C01824=1205.778,287.923,-66.895,-176.683,7.105,148.360
C01825=1205.774,288.171,-66.924,-176.680,7.108,148.360
C01826=1205.769,288.419,-66.953,-176.678,7.110,148.360
C01827=1205.765,288.694,-66.985,-176.675,7.113,148.360
C01828=1205.760,288.968,-67.017,-176.672,7.116,148.360
C01829=1205.756,289.243,-67.049,-176.670,7.119,148.360
C01830=1205.750,289.517,-67.081,-176.667,7.122,148.360
C01831=1205.747,289.765,-67.110,-176.664,7.124,148.359
C01832=1205.742,290.013,-67.139,-176.662,7.127,148.359
C01833=1205.738,290.261,-67.168,-176.660,7.129,148.359
C01834=1205.733,290.510,-67.197,-176.657,7.132,148.359
C01835=1205.729,290.758,-67.226,-176.655,7.134,148.359
C01836=1205.725,291.006,-67.256,-176.652,7.137,148.359
C01837=1205.720,291.255,-67.284,-176.650,7.139,148.359
C01838=1205.715,291.503,-67.314,-176.647,7.142,148.359
C01839=1205.712,291.751,-67.342,-176.645,7.144,148.359
C01840=1205.708,291.999,-67.372,-176.642,7.147,148.359
C01841=1205.703,292.248,-67.401,-176.640,7.149,148.359
C01842=1205.699,292.496,-67.430,-176.637,7.152,148.359
C01843=1205.694,292.744,-67.459,-176.635,7.154,148.359
C01844=1205.690,292.992,-67.489,-176.632,7.158,148.359
C01845=1205.686,293.240,-67.518,-176.630,7.160,148.359
C01846=1205.682,293.489,-67.547,-176.627,7.162,148.358
C01847=1205.677,293.737,-67.576,-176.624,7.165,148.358
C01848=1205.673,293.985,-67.605,-176.622,7.168,148.358
C01849=1205.668,294.233,-67.635,-176.620,7.171,148.358
C01850=1205.664,294.482,-67.664,-176.617,7.173,148.358
C01851=1205.660,294.730,-67.694,-176.615,7.176,148.358
C01852=1205.656,294.978,-67.723,-176.613,7.178,148.358
C01853=1205.651,295.227,-67.752,-176.610,7.181,148.358
C01854=1205.647,295.475,-67.781,-176.608,7.183,148.358
C01855=1205.642,295.723,-67.810,-176.605,7.186,148.358
C01856=1205.638,295.971,-67.840,-176.603,7.189,148.358
C01857=1205.634,296.219,-67.869,-176.600,7.191,148.358
C01858=1205.630,296.468,-67.899,-176.597,7.194,148.358
C01859=1205.626,296.716,-67.928,-176.595,7.196,148.358
C01860=1205.621,296.964,-67.958,-176.592,7.199,148.358
C01861=1205.617,297.213,-67.987,-176.590,7.202,148.357
C01862=1205.613,297.461,-68.017,-176.588,7.205,148.357
C01863=1205.608,297.709,-68.047,-176.585,7.207,148.357
C01864=1205.603,297.957,-68.076,-176.583,7.210,148.357
C01865=1205.599,298.205,-68.105,-176.581,7.212,148.357
C01866=1205.595,298.453,-68.135,-176.578,7.215,148.357
C01867=1205.591,298.702,-68.164,-176.575,7.218,148.357
C01868=1205.587,298.950,-68.194,-176.573,7.220,148.357
C01869=1205.583,299.198,-68.224,-176.570,7.223,148.357
C01870=1205.579,299.446,-68.253,-176.568,7.226,148.357
C01871=1205.574,299.694,-68.283,-176.566,7.229,148.357
C01872=1205.570,299.943,-68.313,-176.563,7.231,148.357
C01873=1205.565,300.191,-68.342,-176.561,7.234,148.357
C01874=1205.561,300.439,-68.372,-176.558,7.237,148.357
C01875=1205.557,300.688,-68.401,-176.556,7.239,148.357
C01876=1205.553,300.935,-68.431,-176.553,7.242,148.357
C01877=1205.548,301.184,-68.461,-176.551,7.244,148.357
C01878=1205.544,301.432,-68.491,-176.548,7.247,148.357
C01879=1205.540,301.680,-68.520,-176.546,7.249,148.357
C01880=1205.536,301.929,-68.550,-176.544,7.252,148.357
C01881=1205.531,302.177,-68.580,-176.541,7.256,148.357
C01882=1205.527,302.425,-68.610,-176.539,7.258,148.357
C01883=1205.523,302.673,-68.639,-176.536,7.261,148.357
C01884=1205.518,302.921,-68.669,-176.534,7.263,148.357
C01885=1205.514,303.169,-68.700,-176.531,7.266,148.357
C01886=1205.510,303.418,-68.729,-176.529,7.268,148.357
C01887=1205.506,303.666,-68.758,-176.526,7.271,148.357
C01888=1205.501,303.914,-68.789,-176.524,7.274,148.357
C01889=1205.497,304.162,-68.819,-176.522,7.276,148.357
C01890=1205.493,304.410,-68.848,-176.519,7.279,148.356
C01891=1205.488,304.658,-68.879,-176.517,7.282,148.356
C01892=1205.484,304.907,-68.908,-176.514,7.285,148.356
C01893=1205.480,305.154,-68.939,-176.511,7.288,148.356
C01894=1205.475,305.403,-68.969,-176.509,7.290,148.356
C01895=1205.471,305.651,-68.998,-176.507,7.293,148.356
C01896=1205.467,305.899,-69.028,-176.505,7.295,148.356
C01897=1205.462,306.147,-69.058,-176.502,7.298,148.356
C01898=1205.458,306.395,-69.088,-176.500,7.301,148.356
C01899=1205.454,306.643,-69.118,-176.497,7.304,148.356
C01900=1205.449,306.891,-69.149,-176.495,7.307,148.356
C01901=1205.445,307.139,-69.178,-176.493,7.309,148.356
C01902=1205.441,307.388,-69.209,-176.490,7.312,148.356
C01903=1205.437,307.636,-69.239,-176.488,7.314,148.356
C01904=1205.433,307.884,-69.269,-176.485,7.317,148.356
C01905=1205.428,308.133,-69.299,-176.482,7.320,148.356
C01906=1205.424,308.380,-69.329,-176.480,7.322,148.356
C01907=1205.419,308.629,-69.359,-176.478,7.325,148.356
C01908=1205.415,308.876,-69.389,-176.475,7.329,148.356
C01909=1205.411,309.125,-69.419,-176.473,7.331,148.356
C01910=1205.407,309.373,-69.449,-176.471,7.334,148.356
C01911=1205.403,309.621,-69.481,-176.469,7.336,148.356
C01912=1205.398,309.870,-69.510,-176.466,7.339,148.356
C01913=1205.394,310.118,-69.541,-176.463,7.342,148.356
C01914=1205.390,310.365,-69.571,-176.461,7.344,148.356
C01915=1205.385,310.614,-69.601,-176.458,7.347,148.356
C01916=1205.381,310.861,-69.631,-176.457,7.350,148.356
C01917=1205.377,311.110,-69.662,-176.454,7.353,148.356
C01918=1205.373,311.358,-69.692,-176.451,7.356,148.356
C01919=1205.368,311.606,-69.723,-176.449,7.358,148.356
C01920=1205.365,311.854,-69.753,-176.446,7.361,148.356
C01921=1205.360,312.103,-69.783,-176.444,7.363,148.356
C01922=1205.356,312.350,-69.813,-176.442,7.367,148.356
C01923=1205.352,312.599,-69.844,-176.439,7.370,148.356
C01924=1205.347,312.847,-69.875,-176.437,7.372,148.356
C01925=1205.343,313.094,-69.905,-176.435,7.375,148.356
C01926=1205.338,313.343,-69.935,-176.432,7.378,148.356
C01927=1205.334,313.591,-69.965,-176.430,7.381,148.357
C01928=1205.330,313.839,-69.996,-176.428,7.384,148.357
C01929=1205.326,314.087,-70.027,-176.425,7.386,148.356
C01930=1205.322,314.335,-70.057,-176.423,7.389,148.356
C01931=1205.317,314.611,-70.091,-176.420,7.392,148.356
C01932=1205.312,314.887,-70.125,-176.418,7.395,148.357
C01933=1205.308,315.164,-70.159,-176.415,7.398,148.357
C01934=1205.303,315.440,-70.193,-176.413,7.401,148.357
C01935=1205.298,315.688,-70.224,-176.410,7.404,148.357
C01936=1205.294,315.936,-70.254,-176.408,7.406,148.357
C01937=1205.290,316.184,-70.285,-176.406,7.410,148.357
C01938=1205.286,316.432,-70.316,-176.403,7.413,148.357
C01939=1205.282,316.680,-70.346,-176.401,7.415,148.357
C01940=1205.277,316.928,-70.377,-176.398,7.418,148.357
C01941=1205.273,317.177,-70.408,-176.396,7.421,148.357
C01942=1205.269,317.424,-70.438,-176.394,7.424,148.357
C01943=1205.265,317.672,-70.469,-176.391,7.427,148.357
C01944=1205.261,317.921,-70.500,-176.389,7.429,148.357
C01945=1205.256,318.169,-70.531,-176.387,7.432,148.357
C01946=1205.252,318.416,-70.561,-176.384,7.435,148.357
C01947=1205.248,318.665,-70.592,-176.382,7.437,148.357
C01948=1205.244,318.913,-70.623,-176.380,7.441,148.357
C01949=1205.239,319.161,-70.654,-176.377,7.444,148.357
C01950=1205.236,319.409,-70.684,-176.375,7.446,148.357
C01951=1205.231,319.657,-70.715,-176.373,7.449,148.357
C01952=1205.226,319.905,-70.746,-176.370,7.452,148.357
C01953=1205.222,320.154,-70.777,-176.368,7.455,148.357
C01954=1205.218,320.401,-70.809,-176.365,7.458,148.357
C01955=1205.214,320.649,-70.839,-176.363,7.460,148.357
C01956=1205.210,320.898,-70.870,-176.361,7.463,148.357
C01957=1205.206,321.145,-70.901,-176.359,7.466,148.358
C01958=1205.201,321.393,-70.931,-176.356,7.469,148.358
C01959=1205.197,321.641,-70.963,-176.354,7.472,148.358
C01960=1205.193,321.889,-70.994,-176.352,7.475,148.358
C01961=1205.188,322.137,-71.025,-176.349,7.477,148.358
C01962=1205.185,322.386,-71.055,-176.347,7.480,148.358
C01963=1205.180,322.633,-71.087,-176.345,7.483,148.358
C01964=1205.176,322.882,-71.118,-176.342,7.486,148.358
C01965=1205.172,323.130,-71.149,-176.340,7.489,148.358
C01966=1205.167,323.378,-71.179,-176.338,7.491,148.358
C01967=1205.164,323.626,-71.211,-176.335,7.494,148.358
C01968=1205.159,323.874,-71.242,-176.333,7.498,148.358
C01969=1205.155,324.122,-71.273,-176.331,7.500,148.358
C01970=1205.151,324.370,-71.305,-176.329,7.503,148.359
C01971=1205.147,324.618,-71.336,-176.326,7.506,148.359
C01972=1205.142,324.866,-71.367,-176.324,7.509,148.358
C01973=1205.138,325.114,-71.398,-176.322,7.512,148.359
C01974=1205.134,325.362,-71.429,-176.319,7.515,148.359
C01975=1205.130,325.609,-71.460,-176.317,7.517,148.359
C01976=1205.126,325.858,-71.491,-176.315,7.520,148.359
C01977=1205.121,326.106,-71.522,-176.313,7.523,148.359
C01978=1205.118,326.354,-71.554,-176.310,7.526,148.359
C01979=1205.113,326.602,-71.585,-176.308,7.529,148.359
C01980=1205.109,326.850,-71.616,-176.306,7.531,148.359
C01981=1205.105,327.098,-71.647,-176.303,7.535,148.359
C01982=1205.100,327.346,-71.679,-176.301,7.538,148.359
C01983=1205.096,327.594,-71.710,-176.299,7.540,148.359
C01984=1205.091,327.842,-71.742,-176.297,7.543,148.360
C01985=1205.087,328.090,-71.773,-176.294,7.546,148.360
C01986=1205.083,328.338,-71.804,-176.293,7.549,148.360
C01987=1205.079,328.586,-71.836,-176.290,7.552,148.360
C01988=1205.075,328.834,-71.867,-176.288,7.555,148.360
C01989=1205.071,329.082,-71.898,-176.285,7.558,148.360
C01990=1205.067,329.330,-71.930,-176.283,7.561,148.360
C01991=1205.063,329.578,-71.961,-176.282,7.563,148.360
C01992=1205.058,329.826,-71.992,-176.279,7.566,148.360
C01993=1205.054,330.074,-72.024,-176.277,7.570,148.361
C01994=1205.050,330.323,-72.056,-176.275,7.572,148.360
C01995=1205.045,330.570,-72.087,-176.272,7.575,148.361
C01996=1205.042,330.818,-72.119,-176.270,7.578,148.361
C01997=1205.037,331.066,-72.150,-176.268,7.581,148.361
C01998=1205.033,331.314,-72.182,-176.265,7.584,148.361
C01999=1205.029,331.561,-72.213,-176.263,7.587,148.361
C02000=1205.025,331.810,-72.244,-176.261,7.590,148.361
C02001=1205.020,332.058,-72.276,-176.259,7.593,148.361
C02002=1205.016,332.306,-72.308,-176.257,7.596,148.362
C02003=1205.012,332.553,-72.340,-176.254,7.598,148.361
C02004=1205.008,332.802,-72.371,-176.252,7.602,148.362
C02005=1205.004,333.050,-72.403,-176.251,7.604,148.362
C02006=1204.999,333.297,-72.435,-176.248,7.607,148.362
C02007=1204.996,333.545,-72.467,-176.246,7.611,148.362
C02008=1204.991,333.793,-72.498,-176.244,7.613,148.362
C02009=1204.987,334.041,-72.529,-176.241,7.616,148.362
C02010=1204.983,334.290,-72.562,-176.239,7.619,148.362
C02011=1204.978,334.537,-72.593,-176.237,7.622,148.362
C02012=1204.975,334.785,-72.625,-176.235,7.625,148.363
C02013=1204.970,335.032,-72.657,-176.233,7.628,148.363
C02014=1204.966,335.281,-72.689,-176.230,7.631,148.363
C02015=1204.962,335.529,-72.720,-176.228,7.634,148.363
C02016=1204.958,335.777,-72.752,-176.226,7.637,148.363
C02017=1204.953,336.025,-72.784,-176.224,7.640,148.363
C02018=1204.950,336.273,-72.816,-176.222,7.643,148.363
C02019=1204.945,336.520,-72.847,-176.220,7.645,148.364
C02020=1204.941,336.769,-72.880,-176.218,7.649,148.364
C02021=1204.936,337.016,-72.911,-176.215,7.652,148.364
C02022=1204.933,337.264,-72.943,-176.213,7.654,148.364
C02023=1204.928,337.513,-72.976,-176.211,7.657,148.364
C02024=1204.924,337.760,-73.007,-176.209,7.661,148.364
C02025=1204.920,338.008,-73.039,-176.207,7.663,148.364
C02026=1204.916,338.256,-73.071,-176.205,7.666,148.365
C02027=1204.912,338.504,-73.103,-176.202,7.670,148.365
C02028=1204.908,338.752,-73.135,-176.201,7.672,148.365
C02029=1204.903,339.000,-73.167,-176.198,7.675,148.365
C02030=1204.900,339.248,-73.199,-176.196,7.678,148.365
C02031=1204.895,339.496,-73.231,-176.194,7.681,148.365
C02032=1204.891,339.744,-73.263,-176.192,7.684,148.366
C02033=1204.887,339.992,-73.295,-176.190,7.687,148.366
C02034=1204.883,340.239,-73.327,-176.188,7.690,148.366
C02035=1204.878,340.518,-73.363,-176.186,7.693,148.366
C02036=1204.873,340.795,-73.399,-176.183,7.697,148.366
C02037=1204.869,341.074,-73.435,-176.181,7.700,148.367
C02038=1204.864,341.353,-73.471,-176.179,7.703,148.367
C02039=1204.860,341.600,-73.504,-176.177,7.707,148.367
C02040=1204.856,341.848,-73.536,-176.174,7.710,148.367
C02041=1204.851,342.096,-73.567,-176.172,7.712,148.367
C02042=1204.847,342.344,-73.600,-176.170,7.716,148.367
C02043=1204.843,342.592,-73.632,-176.168,7.718,148.368
C02044=1204.839,342.840,-73.665,-176.166,7.721,148.368
C02045=1204.835,343.087,-73.696,-176.164,7.725,148.368
C02046=1204.830,343.335,-73.729,-176.162,7.727,148.368
C02047=1204.826,343.584,-73.761,-176.160,7.731,148.368
C02048=1204.823,343.831,-73.794,-176.158,7.734,148.369
C02049=1204.818,344.079,-73.826,-176.156,7.736,148.369
C02050=1204.814,344.327,-73.858,-176.154,7.739,148.369
C02051=1204.810,344.575,-73.891,-176.151,7.743,148.369
C02052=1204.806,344.823,-73.923,-176.150,7.745,148.369
C02053=1204.802,345.071,-73.955,-176.147,7.749,148.369
C02054=1204.797,345.318,-73.988,-176.146,7.751,148.370
C02055=1204.793,345.566,-74.020,-176.144,7.755,148.370
C02056=1204.789,345.814,-74.052,-176.141,7.758,148.370
C02057=1204.785,346.062,-74.085,-176.140,7.760,148.370
C02058=1204.781,346.310,-74.117,-176.137,7.764,148.370
C02059=1204.776,346.557,-74.150,-176.136,7.766,148.371
C02060=1204.772,346.805,-74.182,-176.134,7.770,148.371
C02061=1204.768,347.054,-74.214,-176.131,7.773,148.371
C02062=1204.764,347.301,-74.247,-176.130,7.775,148.371
C02063=1204.760,347.549,-74.279,-176.128,7.779,148.371
C02064=1204.755,347.796,-74.312,-176.125,7.782,148.372
C02065=1204.751,348.045,-74.345,-176.124,7.785,148.372
C02066=1204.747,348.292,-74.377,-176.121,7.788,148.372
C02067=1204.743,348.541,-74.410,-176.120,7.790,148.372
C02068=1204.739,348.788,-74.443,-176.118,7.794,148.373
C02069=1204.735,349.036,-74.475,-176.116,7.797,148.373
C02070=1204.731,349.284,-74.508,-176.114,7.800,148.373
C02071=1204.726,349.532,-74.540,-176.112,7.803,148.373
C02072=1204.723,349.779,-74.572,-176.110,7.806,148.374
C02073=1204.718,350.027,-74.605,-176.108,7.809,148.374
C02074=1204.714,350.275,-74.638,-176.106,7.813,148.374
C02075=1204.710,350.523,-74.671,-176.104,7.815,148.374
C02076=1204.706,350.771,-74.703,-176.102,7.818,148.374
C02077=1204.702,351.019,-74.736,-176.101,7.821,148.375
C02078=1204.698,351.267,-74.769,-176.099,7.825,148.375
C02079=1204.693,351.515,-74.802,-176.096,7.828,148.375
C02080=1204.690,351.762,-74.834,-176.095,7.830,148.375
C02081=1204.685,352.010,-74.866,-176.092,7.834,148.376
C02082=1204.681,352.258,-74.900,-176.091,7.836,148.376
C02083=1204.677,352.505,-74.933,-176.089,7.840,148.376
C02084=1204.672,352.754,-74.965,-176.087,7.843,148.376
C02085=1204.669,353.001,-74.998,-176.085,7.846,148.377
C02086=1204.665,353.249,-75.031,-176.083,7.849,148.377
C02087=1204.661,353.496,-75.064,-176.082,7.852,148.377
C02088=1204.656,353.745,-75.096,-176.079,7.855,148.377
C02089=1204.652,353.993,-75.130,-176.077,7.859,148.378
C02090=1204.648,354.240,-75.163,-176.076,7.861,148.378
C02091=1204.645,354.488,-75.195,-176.074,7.865,148.378
C02092=1204.640,354.736,-75.228,-176.072,7.867,148.379
C02093=1204.636,354.984,-75.261,-176.070,7.871,148.379
C02094=1204.632,355.232,-75.294,-176.068,7.874,148.379
C02095=1204.628,355.479,-75.327,-176.067,7.877,148.379
C02096=1204.624,355.727,-75.360,-176.064,7.880,148.380
C02097=1204.619,355.975,-75.394,-176.063,7.883,148.380
C02098=1204.615,356.223,-75.426,-176.061,7.886,148.380
C02099=1204.611,356.471,-75.459,-176.059,7.889,148.380
C02100=1204.607,356.718,-75.492,-176.057,7.892,148.381
C02101=1204.603,356.966,-75.525,-176.055,7.896,148.381
C02102=1204.599,357.214,-75.558,-176.054,7.898,148.381
C02103=1204.595,357.461,-75.591,-176.052,7.902,148.382
C02104=1204.591,357.709,-75.624,-176.050,7.904,148.382
C02105=1204.587,357.957,-75.657,-176.048,7.908,148.382
C02106=1204.583,358.205,-75.691,-176.047,7.910,148.382
C02107=1204.578,358.452,-75.724,-176.045,7.914,148.383
C02108=1204.574,358.700,-75.757,-176.043,7.917,148.383
C02109=1204.570,358.948,-75.790,-176.041,7.920,148.383
C02110=1204.566,359.195,-75.823,-176.039,7.924,148.384
C02111=1204.562,359.443,-75.856,-176.038,7.926,148.384
C02112=1204.558,359.691,-75.890,-176.036,7.930,148.384
C02113=1204.554,359.939,-75.923,-176.034,7.932,148.385
C02114=1204.549,360.186,-75.956,-176.032,7.936,148.385
C02115=1204.545,360.434,-75.989,-176.031,7.938,148.385
C02116=1204.541,360.682,-76.022,-176.029,7.942,148.386
C02117=1204.537,360.930,-76.055,-176.027,7.945,148.386
C02118=1204.533,361.177,-76.088,-176.026,7.948,148.386
C02119=1204.529,361.425,-76.122,-176.024,7.951,148.386
C02120=1204.525,361.673,-76.155,-176.022,7.954,148.387
C02121=1204.521,361.921,-76.188,-176.021,7.957,148.387
C02122=1204.517,362.169,-76.221,-176.019,7.961,148.387
C02123=1204.513,362.417,-76.255,-176.018,7.963,148.388
C02124=1204.509,362.664,-76.288,-176.015,7.967,148.388
C02125=1204.505,362.912,-76.322,-176.014,7.970,148.388
C02126=1204.500,363.160,-76.355,-176.012,7.973,148.389
C02127=1204.496,363.407,-76.389,-176.011,7.976,148.389
C02128=1204.492,363.655,-76.422,-176.009,7.979,148.390
C02129=1204.488,363.903,-76.455,-176.007,7.982,148.390
C02130=1204.484,364.151,-76.489,-176.006,7.985,148.390
C02131=1204.480,364.398,-76.522,-176.004,7.988,148.391
C02132=1204.476,364.646,-76.555,-176.002,7.992,148.391
C02133=1204.472,364.894,-76.589,-176.001,7.994,148.391
C02134=1204.467,365.141,-76.623,-175.999,7.998,148.392
C02135=1204.463,365.389,-76.656,-175.998,8.001,148.392
C02136=1204.459,365.637,-76.689,-175.996,8.003,148.392
C02137=1204.456,365.885,-76.723,-175.995,8.007,148.393
C02138=1204.452,366.132,-76.757,-175.993,8.010,148.393
C02139=1204.447,366.413,-76.795,-175.992,8.013,148.393
C02140=1204.442,366.693,-76.832,-175.990,8.017,148.394
C02141=1204.437,366.974,-76.871,-175.988,8.021,148.394
C02142=1204.433,367.254,-76.908,-175.986,8.024,148.395
C02143=1204.428,367.502,-76.942,-175.985,8.027,148.395
C02144=1204.424,367.750,-76.975,-175.983,8.031,148.395
C02145=1204.421,367.997,-77.010,-175.982,8.033,148.396
C02146=1204.417,368.245,-77.043,-175.980,8.036,148.396
C02147=1204.412,368.493,-77.077,-175.979,8.040,148.397
C02148=1204.408,368.740,-77.110,-175.977,8.043,148.397
C02149=1204.404,368.988,-77.144,-175.976,8.045,148.397
C02150=1204.401,369.236,-77.178,-175.974,8.049,148.398
C02151=1204.396,369.484,-77.211,-175.973,8.052,148.398
C02152=1204.392,369.731,-77.245,-175.972,8.054,148.398
C02153=1204.388,369.979,-77.279,-175.970,8.058,148.399
C02154=1204.384,370.226,-77.312,-175.969,8.061,148.399
C02155=1204.380,370.475,-77.347,-175.967,8.064,148.400
C02156=1204.376,370.722,-77.380,-175.966,8.067,148.400
C02157=1204.372,370.969,-77.414,-175.964,8.070,148.400
C02158=1204.367,371.217,-77.447,-175.963,8.073,148.401
C02159=1204.364,371.465,-77.482,-175.962,8.076,148.401
C02160=1204.360,371.713,-77.515,-175.960,8.079,148.402
C02161=1204.355,371.960,-77.549,-175.959,8.082,148.402
C02162=1204.351,372.208,-77.583,-175.958,8.085,148.402
C02163=1204.347,372.455,-77.616,-175.956,8.089,148.403
C02164=1204.343,372.703,-77.651,-175.955,8.092,148.404
C02165=1204.339,372.951,-77.684,-175.954,8.095,148.404
C02166=1204.335,373.198,-77.718,-175.953,8.097,148.404
C02167=1204.331,373.447,-77.752,-175.952,8.100,148.405
C02168=1204.327,373.694,-77.786,-175.950,8.104,148.405
C02169=1204.323,373.941,-77.820,-175.949,8.107,148.406
C02170=1204.318,374.189,-77.854,-175.947,8.109,148.406
C02171=1204.315,374.437,-77.888,-175.946,8.112,148.406
C02172=1204.310,374.685,-77.922,-175.945,8.115,148.407
C02173=1204.306,374.932,-77.956,-175.944,8.119,148.407
C02174=1204.303,375.179,-77.989,-175.942,8.122,148.408
C02175=1204.298,375.428,-78.023,-175.941,8.125,148.408
C02176=1204.295,375.675,-78.057,-175.940,8.127,148.408
C02177=1204.290,375.923,-78.092,-175.939,8.130,148.409
C02178=1204.286,376.171,-78.125,-175.938,8.133,148.409
C02179=1204.283,376.418,-78.159,-175.936,8.137,148.410
C02180=1204.278,376.666,-78.194,-175.935,8.140,148.410
C02181=1204.275,376.913,-78.228,-175.934,8.143,148.411
C02182=1204.270,377.161,-78.262,-175.933,8.146,148.411
C02183=1204.266,377.408,-78.296,-175.932,8.148,148.412
C02184=1204.262,377.656,-78.330,-175.931,8.151,148.412
C02185=1204.258,377.904,-78.364,-175.930,8.154,148.413
C02186=1204.253,378.152,-78.398,-175.929,8.157,148.413
C02187=1204.250,378.399,-78.432,-175.928,8.160,148.413
C02188=1204.246,378.647,-78.467,-175.927,8.163,148.414
C02189=1204.242,378.894,-78.501,-175.926,8.166,148.414
C02190=1204.237,379.142,-78.534,-175.924,8.170,148.415
C02191=1204.234,379.390,-78.569,-175.923,8.173,148.415
C02192=1204.229,379.637,-78.603,-175.922,8.175,148.416
C02193=1204.225,379.884,-78.637,-175.921,8.178,148.416
C02194=1204.221,380.133,-78.672,-175.920,8.181,148.417
C02195=1204.217,380.380,-78.705,-175.919,8.184,148.417
C02196=1204.213,380.628,-78.739,-175.918,8.187,148.418
C02197=1204.209,380.876,-78.774,-175.917,8.190,148.418
C02198=1204.205,381.123,-78.808,-175.916,8.193,148.419
C02199=1204.202,381.371,-78.842,-175.915,8.196,148.419
C02200=1204.197,381.618,-78.877,-175.913,8.199,148.420
C02201=1204.193,381.865,-78.911,-175.913,8.201,148.420
C02202=1204.189,382.113,-78.945,-175.912,8.204,148.421
C02203=1204.184,382.361,-78.979,-175.911,8.207,148.421
C02204=1204.180,382.609,-79.013,-175.910,8.210,148.421
C02205=1204.177,382.857,-79.048,-175.909,8.213,148.422
C02206=1204.173,383.104,-79.082,-175.908,8.216,148.422
C02207=1204.169,383.352,-79.117,-175.907,8.219,148.423
C02208=1204.164,383.599,-79.151,-175.906,8.222,148.423
C02209=1204.160,383.846,-79.185,-175.905,8.225,148.424
C02210=1204.156,384.095,-79.220,-175.904,8.228,148.424
C02211=1204.153,384.342,-79.254,-175.904,8.230,148.425
C02212=1204.149,384.590,-79.289,-175.903,8.233,148.425
C02213=1204.144,384.837,-79.323,-175.902,8.236,148.426
C02214=1204.140,385.084,-79.357,-175.901,8.239,148.427
C02215=1204.136,385.332,-79.392,-175.900,8.242,148.427
C02216=1204.132,385.580,-79.426,-175.899,8.245,148.428
C02217=1204.128,385.828,-79.460,-175.898,8.247,148.428
C02218=1204.124,386.075,-79.495,-175.898,8.250,148.428
C02219=1204.120,386.322,-79.529,-175.897,8.253,148.429
C02220=1204.116,386.570,-79.564,-175.896,8.256,148.429
C02221=1204.111,386.818,-79.598,-175.895,8.259,148.430
C02222=1204.108,387.066,-79.632,-175.894,8.261,148.430
C02223=1204.104,387.313,-79.667,-175.894,8.264,148.431
C02224=1204.100,387.561,-79.702,-175.893,8.267,148.432
C02225=1204.096,387.808,-79.735,-175.892,8.269,148.432
C02226=1204.092,388.056,-79.771,-175.891,8.272,148.432
C02227=1204.088,388.303,-79.805,-175.891,8.275,148.433
C02228=1204.084,388.550,-79.839,-175.889,8.278,148.433
C02229=1204.080,388.798,-79.874,-175.889,8.280,148.434
C02230=1204.075,389.046,-79.909,-175.888,8.283,148.435
C02231=1204.072,389.294,-79.943,-175.887,8.286,148.435
C02232=1204.067,389.541,-79.977,-175.887,8.288,148.436
C02233=1204.063,389.789,-80.012,-175.886,8.292,148.436
C02234=1204.059,390.037,-80.047,-175.885,8.295,148.437
C02235=1204.056,390.284,-80.082,-175.885,8.297,148.437
C02236=1204.051,390.531,-80.116,-175.884,8.300,148.438
C02237=1204.047,390.779,-80.151,-175.884,8.302,148.438
C02238=1204.044,391.026,-80.185,-175.883,8.305,148.439
C02239=1204.040,391.275,-80.220,-175.882,8.308,148.439
C02240=1204.035,391.522,-80.254,-175.882,8.310,148.440
C02241=1204.031,391.769,-80.290,-175.881,8.313,148.440
C02242=1204.028,392.017,-80.323,-175.880,8.315,148.441
C02243=1204.022,392.300,-80.363,-175.879,8.318,148.441
C02244=1204.018,392.582,-80.403,-175.879,8.321,148.442
C02245=1204.013,392.865,-80.442,-175.878,8.325,148.442
C02246=1204.009,393.148,-80.482,-175.877,8.328,148.443
C02247=1204.005,393.395,-80.516,-175.877,8.330,148.444
C02248=1204.001,393.642,-80.552,-175.876,8.333,148.444
C02249=1203.997,393.890,-80.586,-175.876,8.335,148.445
C02250=1203.993,394.138,-80.621,-175.875,8.338,148.445
C02251=1203.988,394.385,-80.655,-175.874,8.340,148.446
C02252=1203.985,394.633,-80.691,-175.874,8.344,148.446
C02253=1203.980,394.880,-80.725,-175.873,8.346,148.447
C02254=1203.977,395.128,-80.759,-175.873,8.349,148.447
C02255=1203.972,395.375,-80.794,-175.872,8.351,148.448
C02256=1203.969,395.623,-80.829,-175.871,8.354,148.448
C02257=1203.964,395.870,-80.864,-175.871,8.356,148.449
C02258=1203.960,396.118,-80.899,-175.871,8.359,148.449
C02259=1203.957,396.365,-80.933,-175.870,8.362,148.450
C02260=1203.953,396.613,-80.968,-175.869,8.364,148.450
C02261=1203.949,396.861,-81.003,-175.869,8.367,148.451
C02262=1203.945,397.108,-81.038,-175.868,8.369,148.451
C02263=1203.941,397.356,-81.073,-175.868,8.371,148.452
C02264=1203.936,397.603,-81.107,-175.867,8.374,148.452
C02265=1203.933,397.851,-81.142,-175.867,8.376,148.453
C02266=1203.928,398.098,-81.177,-175.866,8.379,148.453
C02267=1203.925,398.346,-81.212,-175.866,8.382,148.454
C02268=1203.920,398.593,-81.247,-175.865,8.384,148.454
C02269=1203.916,398.841,-81.282,-175.865,8.387,148.455
C02270=1203.912,399.088,-81.317,-175.864,8.389,148.456
C02271=1203.908,399.336,-81.352,-175.864,8.391,148.456
C02272=1203.905,399.584,-81.386,-175.864,8.394,148.456
C02273=1203.901,399.831,-81.421,-175.863,8.397,148.457
C02274=1203.897,400.079,-81.456,-175.863,8.399,148.458
C02275=1203.892,400.325,-81.491,-175.862,8.401,148.458
C02276=1203.888,400.574,-81.526,-175.862,8.404,148.459
C02277=1203.884,400.821,-81.560,-175.861,8.406,148.459
C02278=1203.880,401.068,-81.596,-175.861,8.409,148.460
C02279=1203.876,401.316,-81.630,-175.860,8.411,148.460
C02280=1203.872,401.563,-81.666,-175.860,8.414,148.461
C02281=1203.869,401.811,-81.700,-175.859,8.416,148.461
C02282=1203.864,402.058,-81.735,-175.859,8.418,148.462
C02283=1203.860,402.306,-81.770,-175.859,8.420,148.462
C02284=1203.856,402.553,-81.805,-175.858,8.423,148.463
C02285=1203.852,402.801,-81.840,-175.858,8.426,148.463
C02286=1203.848,403.049,-81.875,-175.857,8.428,148.464
C02287=1203.844,403.296,-81.910,-175.857,8.430,148.464
C02288=1203.840,403.544,-81.945,-175.856,8.432,148.465
C02289=1203.836,403.791,-81.980,-175.856,8.435,148.465
C02290=1203.832,404.039,-82.015,-175.855,8.438,148.466
C02291=1203.827,404.286,-82.050,-175.855,8.440,148.466
C02292=1203.824,404.534,-82.085,-175.855,8.442,148.467
C02293=1203.820,404.781,-82.121,-175.855,8.444,148.467
C02294=1203.816,405.028,-82.156,-175.854,8.446,148.468
C02295=1203.812,405.276,-82.191,-175.854,8.449,148.468
C02296=1203.809,405.524,-82.226,-175.854,8.451,148.469
C02297=1203.804,405.771,-82.260,-175.853,8.454,148.469
C02298=1203.800,406.018,-82.296,-175.853,8.456,148.470
C02299=1203.796,406.266,-82.330,-175.853,8.459,148.470
C02300=1203.792,406.513,-82.366,-175.852,8.461,148.471
C02301=1203.788,406.762,-82.400,-175.852,8.463,148.471
C02302=1203.784,407.008,-82.436,-175.851,8.465,148.472
C02303=1203.780,407.256,-82.470,-175.851,8.467,148.472
C02304=1203.776,407.503,-82.506,-175.851,8.470,148.473
C02305=1203.772,407.751,-82.541,-175.850,8.472,148.473
C02306=1203.768,407.999,-82.576,-175.850,8.474,148.474
C02307=1203.764,408.246,-82.611,-175.850,8.476,148.474
C02308=1203.760,408.494,-82.646,-175.850,8.478,148.475
C02309=1203.756,408.741,-82.682,-175.849,8.481,148.475
C02310=1203.752,408.988,-82.717,-175.848,8.484,148.476
C02311=1203.748,409.236,-82.752,-175.848,8.486,148.476
C02312=1203.744,409.484,-82.787,-175.848,8.488,148.477
C02313=1203.740,409.731,-82.822,-175.847,8.490,148.477
C02314=1203.736,409.979,-82.857,-175.847,8.493,148.478
C02315=1203.732,410.225,-82.892,-175.847,8.495,148.478
C02316=1203.728,410.474,-82.927,-175.846,8.497,148.479
C02317=1203.724,410.721,-82.963,-175.846,8.499,148.479
C02318=1203.720,410.968,-82.998,-175.846,8.501,148.480
C02319=1203.716,411.216,-83.033,-175.846,8.504,148.480
C02320=1203.712,411.463,-83.068,-175.845,8.506,148.481
C02321=1203.708,411.710,-83.103,-175.845,8.508,148.481
C02322=1203.704,411.958,-83.138,-175.845,8.510,148.482
C02323=1203.700,412.206,-83.174,-175.845,8.512,148.482
C02324=1203.696,412.453,-83.209,-175.844,8.514,148.482
C02325=1203.691,412.701,-83.244,-175.844,8.516,148.483
C02326=1203.688,412.949,-83.280,-175.844,8.518,148.484
C02327=1203.684,413.195,-83.315,-175.844,8.520,148.484
C02328=1203.680,413.444,-83.350,-175.843,8.522,148.484
C02329=1203.676,413.691,-83.386,-175.843,8.525,148.485
C02330=1203.672,413.938,-83.421,-175.842,8.527,148.485
C02331=1203.668,414.185,-83.456,-175.842,8.529,148.486
C02332=1203.664,414.433,-83.491,-175.842,8.531,148.486
C02333=1203.660,414.680,-83.526,-175.841,8.533,148.487
C02334=1203.656,414.928,-83.562,-175.841,8.536,148.487
C02335=1203.652,415.176,-83.597,-175.841,8.538,148.488
C02336=1203.648,415.423,-83.632,-175.840,8.540,148.488
C02337=1203.644,415.670,-83.667,-175.841,8.541,148.489
C02338=1203.641,415.918,-83.703,-175.840,8.544,148.489
C02339=1203.635,416.213,-83.745,-175.840,8.547,148.490
C02340=1203.632,416.508,-83.787,-175.839,8.549,148.490
C02341=1203.630,416.803,-83.829,-175.839,8.551,148.491
C02342=1203.632,417.097,-83.870,-175.839,8.553,148.491
C02343=1203.210,417.098,-83.909,-175.842,8.564,148.495
C02344=1203.209,416.801,-83.866,-175.842,8.562,148.495
C02345=1203.209,416.503,-83.825,-175.842,8.560,148.494
C02346=1203.214,416.205,-83.782,-175.843,8.557,148.494
C02347=1203.219,415.907,-83.739,-175.844,8.554,148.493
C02348=1203.222,415.659,-83.704,-175.844,8.552,148.492
C02349=1203.226,415.412,-83.668,-175.843,8.550,148.492
C02350=1203.230,415.165,-83.633,-175.844,8.549,148.492
C02351=1203.234,414.917,-83.598,-175.844,8.546,148.491
C02352=1203.238,414.669,-83.563,-175.845,8.544,148.491
C02353=1203.242,414.423,-83.527,-175.845,8.542,148.490
C02354=1203.246,414.175,-83.493,-175.845,8.540,148.490
C02355=1203.250,413.927,-83.457,-175.846,8.537,148.489
C02356=1203.254,413.680,-83.422,-175.846,8.535,148.489
C02357=1203.259,413.432,-83.386,-175.846,8.533,148.488
C02358=1203.263,413.184,-83.351,-175.846,8.531,148.488
C02359=1203.267,412.938,-83.316,-175.847,8.529,148.487
C02360=1203.270,412.690,-83.280,-175.847,8.526,148.487
C02361=1203.274,412.442,-83.245,-175.847,8.525,148.486
C02362=1203.279,412.195,-83.210,-175.847,8.523,148.486
C02363=1203.282,411.948,-83.175,-175.848,8.521,148.485
C02364=1203.286,411.699,-83.140,-175.848,8.519,148.485
C02365=1203.291,411.453,-83.105,-175.848,8.516,148.484
C02366=1203.294,411.205,-83.069,-175.848,8.514,148.484
C02367=1203.298,410.957,-83.034,-175.849,8.512,148.483
C02368=1203.302,410.710,-82.999,-175.849,8.510,148.483
C02369=1203.306,410.463,-82.964,-175.850,8.507,148.482
C02370=1203.310,410.215,-82.929,-175.850,8.505,148.482
C02371=1203.314,409.968,-82.894,-175.850,8.503,148.481
C02372=1203.318,409.720,-82.858,-175.850,8.501,148.481
C02373=1203.322,409.472,-82.823,-175.851,8.499,148.480
C02374=1203.326,409.225,-82.788,-175.851,8.496,148.480
C02375=1203.330,408.978,-82.752,-175.851,8.494,148.479
C02376=1203.334,408.730,-82.718,-175.852,8.492,148.479
C02377=1203.338,408.483,-82.682,-175.852,8.490,148.478
C02378=1203.342,408.235,-82.648,-175.853,8.488,148.478
C02379=1203.346,407.988,-82.612,-175.853,8.485,148.477
C02380=1203.350,407.741,-82.577,-175.854,8.482,148.477
C02381=1203.354,407.492,-82.542,-175.854,8.480,148.476
C02382=1203.358,407.246,-82.507,-175.854,8.478,148.476
C02383=1203.362,406.998,-82.472,-175.854,8.475,148.475
C02384=1203.366,406.750,-82.436,-175.855,8.474,148.475
C02385=1203.370,406.503,-82.401,-175.855,8.471,148.474
C02386=1203.374,406.255,-82.366,-175.855,8.469,148.474
C02387=1203.378,406.008,-82.331,-175.856,8.467,148.473
C02388=1203.382,405.760,-82.296,-175.856,8.464,148.473
C02389=1203.386,405.513,-82.261,-175.856,8.462,148.472
C02390=1203.391,405.265,-82.226,-175.857,8.460,148.472
C02391=1203.394,405.018,-82.191,-175.857,8.457,148.471
C02392=1203.399,404.770,-82.156,-175.858,8.455,148.471
C02393=1203.403,404.523,-82.121,-175.858,8.453,148.470
C02394=1203.406,404.275,-82.086,-175.858,8.450,148.470
C02395=1203.411,404.028,-82.051,-175.859,8.448,148.469
C02396=1203.415,403.780,-82.016,-175.859,8.446,148.469
C02397=1203.419,403.533,-81.981,-175.860,8.443,148.468
C02398=1203.422,403.286,-81.946,-175.860,8.441,148.468
C02399=1203.426,403.038,-81.911,-175.860,8.438,148.467
C02400=1203.430,402.790,-81.877,-175.860,8.436,148.467
C02401=1203.434,402.543,-81.841,-175.861,8.434,148.466
C02402=1203.439,402.295,-81.807,-175.861,8.432,148.466
C02403=1203.442,402.048,-81.771,-175.862,8.429,148.465
C02404=1203.446,401.800,-81.736,-175.862,8.427,148.465
C02405=1203.451,401.553,-81.701,-175.863,8.424,148.464
C02406=1203.455,401.305,-81.666,-175.863,8.422,148.464
C02407=1203.459,401.058,-81.631,-175.864,8.419,148.463
C02408=1203.463,400.810,-81.596,-175.864,8.417,148.463
C02409=1203.467,400.563,-81.561,-175.864,8.415,148.462
C02410=1203.470,400.315,-81.527,-175.865,8.412,148.462
C02411=1203.474,400.067,-81.492,-175.865,8.409,148.461
C02412=1203.478,399.820,-81.457,-175.866,8.407,148.461
C02413=1203.482,399.572,-81.422,-175.866,8.405,148.460
C02414=1203.487,399.325,-81.387,-175.867,8.402,148.460
C02415=1203.491,399.077,-81.352,-175.867,8.400,148.459
C02416=1203.495,398.831,-81.317,-175.868,8.397,148.459
C02417=1203.499,398.582,-81.282,-175.868,8.395,148.458
C02418=1203.502,398.335,-81.248,-175.869,8.392,148.457
C02419=1203.506,398.088,-81.212,-175.869,8.390,148.457
C02420=1203.510,397.840,-81.178,-175.870,8.387,148.457
C02421=1203.515,397.592,-81.143,-175.870,8.385,148.456
C02422=1203.519,397.345,-81.108,-175.870,8.382,148.455
C02423=1203.523,397.097,-81.073,-175.871,8.379,148.455
C02424=1203.527,396.849,-81.038,-175.871,8.377,148.454
C02425=1203.531,396.603,-81.004,-175.872,8.375,148.454
C02426=1203.535,396.355,-80.969,-175.873,8.372,148.453
C02427=1203.539,396.107,-80.934,-175.873,8.370,148.453
C02428=1203.543,395.860,-80.899,-175.874,8.367,148.452
C02429=1203.547,395.612,-80.864,-175.874,8.364,148.452
C02430=1203.551,395.364,-80.830,-175.874,8.362,148.451
C02431=1203.555,395.118,-80.795,-175.875,8.359,148.451
C02432=1203.559,394.870,-80.760,-175.876,8.357,148.450
C02433=1203.563,394.622,-80.726,-175.876,8.354,148.450
C02434=1203.567,394.375,-80.690,-175.877,8.352,148.449
C02435=1203.571,394.127,-80.655,-175.877,8.349,148.449
C02436=1203.575,393.879,-80.621,-175.878,8.347,148.448
C02437=1203.579,393.631,-80.587,-175.879,8.343,148.448
C02438=1203.583,393.385,-80.551,-175.879,8.341,148.447
C02439=1203.587,393.136,-80.517,-175.880,8.338,148.446
C02440=1203.592,392.853,-80.477,-175.881,8.335,148.446
C02441=1203.596,392.571,-80.438,-175.881,8.332,148.445
C02442=1203.601,392.289,-80.398,-175.882,8.330,148.445
C02443=1203.605,392.006,-80.359,-175.882,8.326,148.444
C02444=1203.609,391.758,-80.324,-175.883,8.323,148.444
C02445=1203.614,391.511,-80.290,-175.884,8.321,148.443
C02446=1203.618,391.263,-80.254,-175.885,8.318,148.443
C02447=1203.622,391.016,-80.220,-175.885,8.315,148.442
C02448=1203.625,390.768,-80.186,-175.886,8.313,148.442
C02449=1203.630,390.521,-80.151,-175.887,8.310,148.441
C02450=1203.634,390.273,-80.116,-175.887,8.308,148.441
C02451=1203.638,390.026,-80.082,-175.888,8.305,148.440
C02452=1203.642,389.778,-80.047,-175.889,8.302,148.440
C02453=1203.646,389.531,-80.012,-175.889,8.300,148.439
C02454=1203.650,389.282,-79.978,-175.890,8.297,148.439
C02455=1203.654,389.035,-79.944,-175.891,8.293,148.438
C02456=1203.658,388.787,-79.909,-175.891,8.291,148.438
C02457=1203.662,388.540,-79.874,-175.892,8.288,148.437
C02458=1203.665,388.293,-79.839,-175.893,8.285,148.436
C02459=1203.670,388.045,-79.805,-175.894,8.283,148.436
C02460=1203.674,387.798,-79.770,-175.894,8.280,148.435
C02461=1203.678,387.550,-79.736,-175.895,8.277,148.435
C02462=1203.682,387.303,-79.702,-175.896,8.274,148.434
C02463=1203.686,387.054,-79.667,-175.897,8.272,148.434
C02464=1203.690,386.807,-79.633,-175.897,8.269,148.433
C02465=1203.694,386.559,-79.598,-175.899,8.266,148.433
C02466=1203.699,386.312,-79.564,-175.899,8.263,148.432
C02467=1203.702,386.064,-79.530,-175.900,8.261,148.432
C02468=1203.706,385.817,-79.495,-175.901,8.258,148.431
C02469=1203.711,385.569,-79.461,-175.902,8.255,148.431
C02470=1203.714,385.321,-79.426,-175.903,8.252,148.430
C02471=1203.719,385.074,-79.392,-175.904,8.249,148.430
C02472=1203.723,384.826,-79.357,-175.905,8.246,148.429
C02473=1203.727,384.579,-79.323,-175.905,8.244,148.429
C02474=1203.731,384.331,-79.289,-175.906,8.241,148.428
C02475=1203.734,384.083,-79.254,-175.907,8.238,148.428
C02476=1203.739,383.836,-79.220,-175.908,8.235,148.427
C02477=1203.743,383.588,-79.185,-175.909,8.232,148.427
C02478=1203.747,383.341,-79.151,-175.910,8.229,148.426
C02479=1203.751,383.093,-79.117,-175.911,8.226,148.426
C02480=1203.755,382.846,-79.083,-175.912,8.223,148.425
C02481=1203.759,382.598,-79.048,-175.912,8.221,148.425
C02482=1203.763,382.350,-79.013,-175.913,8.218,148.424
C02483=1203.767,382.103,-78.979,-175.914,8.215,148.424
C02484=1203.772,381.856,-78.945,-175.915,8.212,148.423
C02485=1203.775,381.608,-78.911,-175.916,8.209,148.423
C02486=1203.779,381.360,-78.876,-175.917,8.206,148.423
C02487=1203.783,381.113,-78.843,-175.918,8.203,148.422
C02488=1203.787,380.864,-78.808,-175.919,8.200,148.422
C02489=1203.791,380.617,-78.774,-175.920,8.197,148.421
C02490=1203.795,380.369,-78.740,-175.921,8.195,148.421
C02491=1203.799,380.122,-78.706,-175.922,8.191,148.420
C02492=1203.804,379.875,-78.671,-175.923,8.189,148.420
C02493=1203.808,379.627,-78.636,-175.924,8.186,148.419
C02494=1203.812,379.379,-78.603,-175.925,8.183,148.419
C02495=1203.816,379.131,-78.569,-175.927,8.180,148.418
C02496=1203.820,378.884,-78.535,-175.927,8.177,148.418
C02497=1203.824,378.636,-78.500,-175.929,8.174,148.417
C02498=1203.828,378.389,-78.466,-175.930,8.171,148.417
C02499=1203.832,378.140,-78.432,-175.931,8.168,148.416
C02500=1203.836,377.893,-78.398,-175.932,8.164,148.416
C02501=1203.841,377.646,-78.364,-175.934,8.162,148.416
C02502=1203.844,377.398,-78.330,-175.934,8.159,148.415
C02503=1203.848,377.150,-78.296,-175.936,8.156,148.415
C02504=1203.853,376.903,-78.262,-175.937,8.153,148.414
C02505=1203.856,376.655,-78.228,-175.938,8.150,148.414
C02506=1203.860,376.408,-78.193,-175.939,8.147,148.413
C02507=1203.864,376.160,-78.160,-175.940,8.144,148.413
C02508=1203.869,375.912,-78.126,-175.942,8.141,148.412
C02509=1203.872,375.665,-78.091,-175.943,8.138,148.412
C02510=1203.877,375.417,-78.058,-175.944,8.135,148.411
C02511=1203.881,375.170,-78.024,-175.945,8.132,148.411
C02512=1203.884,374.922,-77.989,-175.946,8.129,148.411
C02513=1203.889,374.674,-77.956,-175.947,8.126,148.410
C02514=1203.893,374.427,-77.922,-175.949,8.123,148.410
C02515=1203.898,374.179,-77.887,-175.950,8.119,148.409
C02516=1203.901,373.931,-77.854,-175.951,8.117,148.409
C02517=1203.905,373.684,-77.820,-175.952,8.114,148.408
C02518=1203.910,373.436,-77.786,-175.954,8.111,148.408
C02519=1203.913,373.188,-77.752,-175.955,8.107,148.408
C02520=1203.917,372.941,-77.718,-175.957,8.105,148.407
C02521=1203.922,372.693,-77.684,-175.958,8.102,148.407
C02522=1203.926,372.445,-77.651,-175.959,8.099,148.406
C02523=1203.929,372.197,-77.617,-175.961,8.095,148.406
C02524=1203.934,371.950,-77.583,-175.962,8.093,148.406
C02525=1203.938,371.702,-77.549,-175.963,8.089,148.405
C02526=1203.942,371.455,-77.515,-175.964,8.086,148.405
C02527=1203.946,371.206,-77.481,-175.966,8.083,148.404
C02528=1203.950,370.959,-77.448,-175.967,8.080,148.404
C02529=1203.954,370.711,-77.414,-175.968,8.077,148.403
C02530=1203.958,370.464,-77.380,-175.970,8.074,148.403
C02531=1203.963,370.216,-77.347,-175.971,8.071,148.403
C02532=1203.966,369.968,-77.312,-175.972,8.068,148.402
C02533=1203.971,369.720,-77.279,-175.975,8.065,148.402
C02534=1203.974,369.473,-77.245,-175.976,8.062,148.402
C02535=1203.979,369.225,-77.212,-175.977,8.059,148.401
C02536=1203.982,368.978,-77.177,-175.979,8.056,148.401
C02537=1203.987,368.730,-77.144,-175.980,8.053,148.400
C02538=1203.991,368.482,-77.110,-175.981,8.050,148.400
C02539=1203.995,368.235,-77.077,-175.983,8.046,148.400
C02540=1203.999,367.987,-77.044,-175.984,8.043,148.399
C02541=1204.003,367.740,-77.009,-175.986,8.040,148.399
C02542=1204.007,367.491,-76.976,-175.987,8.037,148.398
C02543=1204.011,367.243,-76.942,-175.989,8.034,148.398
C02544=1204.016,366.963,-76.904,-175.990,8.031,148.398
C02545=1204.020,366.682,-76.866,-175.992,8.027,148.397
C02546=1204.025,366.403,-76.828,-175.994,8.024,148.397
C02547=1204.029,366.122,-76.791,-175.996,8.020,148.396
C02548=1204.034,365.874,-76.756,-175.997,8.017,148.396
C02549=1204.038,365.626,-76.723,-175.999,8.013,148.396
C02550=1204.042,365.378,-76.690,-176.000,8.011,148.395
C02551=1204.046,365.131,-76.656,-176.002,8.007,148.395
C02552=1204.050,364.883,-76.623,-176.003,8.005,148.395
C02553=1204.054,364.635,-76.589,-176.005,8.002,148.394
C02554=1204.059,364.387,-76.556,-176.007,7.998,148.394
C02555=1204.063,364.140,-76.522,-176.008,7.996,148.394
C02556=1204.066,363.892,-76.488,-176.010,7.992,148.393
C02557=1204.070,363.644,-76.455,-176.011,7.989,148.393
C02558=1204.074,363.396,-76.422,-176.013,7.986,148.392
C02559=1204.078,363.149,-76.389,-176.014,7.983,148.392
C02560=1204.082,362.902,-76.355,-176.017,7.980,148.392
C02561=1204.086,362.654,-76.322,-176.018,7.977,148.391
C02562=1204.091,362.406,-76.289,-176.020,7.973,148.391
C02563=1204.095,362.158,-76.255,-176.021,7.971,148.391
C02564=1204.099,361.911,-76.222,-176.023,7.967,148.390
C02565=1204.103,361.662,-76.188,-176.025,7.964,148.390
C02566=1204.107,361.414,-76.155,-176.026,7.961,148.390
C02567=1204.111,361.166,-76.122,-176.028,7.958,148.390
C02568=1204.115,360.919,-76.088,-176.030,7.955,148.389
C02569=1204.119,360.672,-76.055,-176.032,7.952,148.389
C02570=1204.124,360.424,-76.022,-176.033,7.949,148.389
C02571=1204.128,360.176,-75.989,-176.035,7.946,148.388
C02572=1204.132,359.928,-75.955,-176.037,7.942,148.388
C02573=1204.136,359.681,-75.922,-176.039,7.939,148.387
C02574=1204.140,359.433,-75.889,-176.040,7.936,148.387
C02575=1204.144,359.185,-75.856,-176.042,7.933,148.387
C02576=1204.148,358.938,-75.823,-176.044,7.930,148.387
C02577=1204.152,358.690,-75.790,-176.046,7.927,148.386
C02578=1204.157,358.442,-75.756,-176.047,7.924,148.386
C02579=1204.161,358.194,-75.723,-176.049,7.921,148.386
C02580=1204.165,357.947,-75.690,-176.050,7.918,148.385
C02581=1204.169,357.699,-75.657,-176.053,7.914,148.385
C02582=1204.173,357.451,-75.624,-176.055,7.911,148.385
C02583=1204.177,357.203,-75.591,-176.056,7.908,148.385
C02584=1204.181,356.955,-75.559,-176.058,7.905,148.384
C02585=1204.185,356.707,-75.525,-176.060,7.902,148.384
C02586=1204.189,356.459,-75.492,-176.062,7.899,148.384
C02587=1204.193,356.212,-75.459,-176.064,7.895,148.383
C02588=1204.197,355.964,-75.426,-176.065,7.893,148.383
C02589=1204.202,355.717,-75.393,-176.067,7.889,148.383
C02590=1204.206,355.469,-75.360,-176.069,7.887,148.383
C02591=1204.210,355.221,-75.327,-176.071,7.883,148.382
C02592=1204.214,354.973,-75.294,-176.072,7.881,148.382
C02593=1204.219,354.725,-75.261,-176.075,7.877,148.382
C02594=1204.222,354.478,-75.229,-176.077,7.874,148.382
C02595=1204.226,354.230,-75.195,-176.078,7.871,148.381
C02596=1204.230,353.982,-75.162,-176.080,7.868,148.381
C02597=1204.235,353.734,-75.130,-176.082,7.865,148.381
C02598=1204.239,353.486,-75.097,-176.084,7.862,148.380
C02599=1204.243,353.239,-75.063,-176.086,7.858,148.380
C02600=1204.247,352.991,-75.032,-176.088,7.856,148.380
C02601=1204.251,352.743,-74.998,-176.090,7.852,148.380
C02602=1204.255,352.495,-74.965,-176.092,7.850,148.380
C02603=1204.259,352.247,-74.932,-176.093,7.846,148.379
C02604=1204.264,351.999,-74.900,-176.096,7.843,148.379
C02605=1204.268,351.751,-74.867,-176.097,7.840,148.379
C02606=1204.271,351.504,-74.834,-176.099,7.837,148.379
C02607=1204.276,351.255,-74.802,-176.101,7.835,148.378
C02608=1204.280,351.008,-74.769,-176.103,7.831,148.378
C02609=1204.284,350.761,-74.736,-176.105,7.828,148.378
C02610=1204.288,350.513,-74.704,-176.107,7.825,148.378
C02611=1204.292,350.265,-74.671,-176.109,7.822,148.377
C02612=1204.297,350.017,-74.638,-176.111,7.818,148.377
C02613=1204.301,349.769,-74.605,-176.113,7.816,148.377
C02614=1204.305,349.521,-74.573,-176.115,7.813,148.377
C02615=1204.309,349.273,-74.540,-176.117,7.810,148.376
C02616=1204.313,349.025,-74.507,-176.119,7.807,148.376
C02617=1204.317,348.778,-74.475,-176.121,7.803,148.376
C02618=1204.321,348.530,-74.442,-176.122,7.801,148.376
C02619=1204.326,348.282,-74.410,-176.125,7.797,148.375
C02620=1204.330,348.034,-74.377,-176.126,7.795,148.375
C02621=1204.334,347.786,-74.345,-176.128,7.791,148.375
C02622=1204.338,347.538,-74.312,-176.131,7.788,148.375
C02623=1204.343,347.291,-74.280,-176.132,7.786,148.375
C02624=1204.346,347.043,-74.248,-176.135,7.782,148.374
C02625=1204.351,346.795,-74.215,-176.137,7.779,148.374
C02626=1204.354,346.547,-74.183,-176.138,7.776,148.374
C02627=1204.358,346.299,-74.150,-176.141,7.773,148.374
C02628=1204.363,346.051,-74.117,-176.142,7.771,148.374
C02629=1204.367,345.804,-74.085,-176.144,7.767,148.373
C02630=1204.371,345.556,-74.052,-176.147,7.764,148.373
C02631=1204.376,345.308,-74.020,-176.148,7.761,148.373
C02632=1204.379,345.060,-73.987,-176.151,7.758,148.373
C02633=1204.384,344.812,-73.955,-176.153,7.755,148.372
C02634=1204.388,344.564,-73.924,-176.154,7.752,148.372
C02635=1204.392,344.317,-73.890,-176.157,7.749,148.372
C02636=1204.396,344.069,-73.859,-176.159,7.745,148.372
C02637=1204.400,343.820,-73.826,-176.161,7.743,148.372
C02638=1204.405,343.573,-73.793,-176.163,7.740,148.371
C02639=1204.409,343.325,-73.761,-176.165,7.737,148.372
C02640=1204.413,343.077,-73.729,-176.167,7.734,148.371
C02641=1204.417,342.829,-73.697,-176.169,7.731,148.371
C02642=1204.421,342.581,-73.664,-176.171,7.728,148.371
C02643=1204.425,342.334,-73.633,-176.173,7.725,148.371
C02644=1204.430,342.085,-73.600,-176.175,7.722,148.370
C02645=1204.433,341.837,-73.568,-176.177,7.719,148.370
C02646=1204.438,341.590,-73.536,-176.179,7.716,148.370
C02647=1204.442,341.342,-73.504,-176.182,7.713,148.370
C02648=1204.447,341.063,-73.468,-176.184,7.709,148.370
C02649=1204.452,340.785,-73.432,-176.186,7.706,148.370
C02650=1204.456,340.507,-73.395,-176.189,7.703,148.369
C02651=1204.460,340.229,-73.359,-176.191,7.699,148.369
C02652=1204.465,339.981,-73.327,-176.193,7.696,148.369
C02653=1204.469,339.733,-73.295,-176.195,7.694,148.369
C02654=1204.474,339.485,-73.263,-176.197,7.690,148.369
C02655=1204.477,339.237,-73.231,-176.199,7.688,148.369
C02656=1204.481,338.989,-73.199,-176.201,7.685,148.368
C02657=1204.486,338.741,-73.167,-176.204,7.682,148.368
C02658=1204.490,338.493,-73.135,-176.206,7.679,148.368
C02659=1204.494,338.245,-73.103,-176.208,7.676,148.368
C02660=1204.499,337.998,-73.072,-176.210,7.672,148.368
C02661=1204.502,337.750,-73.040,-176.212,7.670,148.368
C02662=1204.507,337.501,-73.007,-176.214,7.667,148.368
C02663=1204.511,337.254,-72.976,-176.217,7.663,148.367
C02664=1204.515,337.006,-72.944,-176.218,7.661,148.367
C02665=1204.519,336.758,-72.911,-176.221,7.658,148.367
C02666=1204.523,336.510,-72.880,-176.223,7.655,148.367
C02667=1204.527,336.262,-72.848,-176.225,7.652,148.367
C02668=1204.532,336.014,-72.816,-176.227,7.649,148.367
C02669=1204.536,335.767,-72.784,-176.229,7.646,148.367
C02670=1204.540,335.518,-72.752,-176.231,7.643,148.366
C02671=1204.544,335.270,-72.720,-176.234,7.640,148.366
C02672=1204.548,335.023,-72.688,-176.236,7.638,148.366
C02673=1204.552,334.774,-72.657,-176.238,7.634,148.366
C02674=1204.557,334.527,-72.626,-176.240,7.631,148.366
C02675=1204.561,334.278,-72.593,-176.242,7.629,148.366
C02676=1204.565,334.030,-72.562,-176.245,7.625,148.366
C02677=1204.569,333.783,-72.530,-176.247,7.622,148.365
C02678=1204.573,333.535,-72.498,-176.249,7.620,148.365
C02679=1204.578,333.287,-72.467,-176.251,7.617,148.365
C02680=1204.582,333.039,-72.435,-176.253,7.613,148.365
C02681=1204.586,332.791,-72.403,-176.255,7.611,148.365
C02682=1204.590,332.543,-72.372,-176.258,7.608,148.365
C02683=1204.595,332.294,-72.340,-176.260,7.605,148.365
C02684=1204.599,332.047,-72.309,-176.262,7.602,148.365
C02685=1204.603,331.799,-72.277,-176.264,7.599,148.364
C02686=1204.607,331.552,-72.245,-176.267,7.596,148.364
C02687=1204.611,331.303,-72.214,-176.269,7.593,148.364
C02688=1204.615,331.056,-72.183,-176.271,7.590,148.364
C02689=1204.620,330.807,-72.150,-176.273,7.588,148.364
C02690=1204.624,330.559,-72.119,-176.276,7.585,148.364
C02691=1204.628,330.311,-72.088,-176.278,7.581,148.364
C02692=1204.632,330.063,-72.056,-176.279,7.579,148.364
C02693=1204.636,329.815,-72.025,-176.282,7.576,148.364
C02694=1204.640,329.567,-71.993,-176.284,7.572,148.363
C02695=1204.645,329.319,-71.962,-176.286,7.570,148.363
C02696=1204.648,329.071,-71.930,-176.289,7.567,148.363
C02697=1204.653,328.824,-71.898,-176.291,7.564,148.363
C02698=1204.657,328.575,-71.867,-176.293,7.561,148.363
C02699=1204.662,328.328,-71.836,-176.296,7.558,148.363
C02700=1204.666,328.079,-71.805,-176.298,7.555,148.363
C02701=1204.670,327.832,-71.773,-176.300,7.553,148.363
C02702=1204.674,327.583,-71.742,-176.302,7.549,148.363
C02703=1204.678,327.336,-71.711,-176.305,7.546,148.363
C02704=1204.682,327.087,-71.679,-176.307,7.544,148.363
C02705=1204.687,326.840,-71.648,-176.309,7.541,148.363
C02706=1204.691,326.591,-71.617,-176.311,7.537,148.362
C02707=1204.695,326.344,-71.585,-176.314,7.535,148.362
C02708=1204.700,326.096,-71.555,-176.316,7.532,148.362
C02709=1204.703,325.848,-71.523,-176.318,7.530,148.362
C02710=1204.708,325.600,-71.492,-176.320,7.526,148.362
C02711=1204.712,325.351,-71.461,-176.323,7.523,148.362
C02712=1204.716,325.104,-71.429,-176.325,7.521,148.362
C02713=1204.720,324.855,-71.398,-176.327,7.518,148.362
C02714=1204.725,324.608,-71.367,-176.330,7.515,148.362
C02715=1204.729,324.359,-71.336,-176.332,7.512,148.362
C02716=1204.733,324.111,-71.305,-176.334,7.509,148.362
C02717=1204.738,323.864,-71.273,-176.336,7.506,148.361
C02718=1204.742,323.615,-71.242,-176.339,7.504,148.361
C02719=1204.745,323.367,-71.212,-176.341,7.501,148.361
C02720=1204.749,323.119,-71.180,-176.343,7.497,148.361
C02721=1204.754,322.871,-71.149,-176.346,7.495,148.361
C02722=1204.758,322.624,-71.119,-176.348,7.492,148.361
C02723=1204.762,322.375,-71.088,-176.350,7.489,148.361
C02724=1204.767,322.128,-71.056,-176.353,7.487,148.361
C02725=1204.771,321.879,-71.025,-176.355,7.483,148.361
C02726=1204.775,321.631,-70.994,-176.357,7.481,148.361
C02727=1204.780,321.383,-70.963,-176.360,7.478,148.361
C02728=1204.783,321.135,-70.932,-176.362,7.475,148.361
C02729=1204.788,320.887,-70.901,-176.364,7.472,148.361
C02730=1204.792,320.639,-70.871,-176.367,7.469,148.361
C02731=1204.796,320.391,-70.840,-176.369,7.466,148.361
C02732=1204.801,320.143,-70.809,-176.371,7.464,148.361
C02733=1204.805,319.895,-70.779,-176.374,7.461,148.361
C02734=1204.809,319.646,-70.747,-176.376,7.458,148.360
C02735=1204.813,319.399,-70.716,-176.378,7.455,148.360
C02736=1204.818,319.151,-70.685,-176.381,7.452,148.360
C02737=1204.822,318.902,-70.654,-176.382,7.450,148.360
C02738=1204.825,318.655,-70.624,-176.385,7.447,148.360
C02739=1204.830,318.407,-70.593,-176.388,7.444,148.360
C02740=1204.834,318.158,-70.562,-176.389,7.441,148.360
C02741=1204.839,317.910,-70.531,-176.392,7.438,148.360
C02742=1204.843,317.663,-70.501,-176.395,7.435,148.360
C02743=1204.847,317.414,-70.470,-176.397,7.433,148.360
C02744=1204.851,317.166,-70.439,-176.399,7.430,148.360
C02745=1204.856,316.918,-70.408,-176.402,7.427,148.360
C02746=1204.859,316.670,-70.378,-176.404,7.424,148.360
C02747=1204.864,316.422,-70.347,-176.407,7.421,148.360
C02748=1204.868,316.174,-70.316,-176.408,7.419,148.360
C02749=1204.872,315.926,-70.286,-176.411,7.416,148.360
C02750=1204.876,315.677,-70.255,-176.414,7.413,148.360
C02751=1204.881,315.429,-70.224,-176.416,7.411,148.360
C02752=1204.886,315.153,-70.191,-176.418,7.407,148.360
C02753=1204.891,314.877,-70.156,-176.421,7.404,148.360
C02754=1204.895,314.601,-70.122,-176.423,7.401,148.360
C02755=1204.899,314.325,-70.089,-176.427,7.397,148.360
C02756=1204.904,314.077,-70.058,-176.429,7.395,148.360
C02757=1204.908,313.829,-70.027,-176.431,7.392,148.360
C02758=1204.912,313.581,-69.997,-176.433,7.390,148.360
C02759=1204.917,313.332,-69.967,-176.436,7.387,148.360
C02760=1204.921,313.084,-69.936,-176.438,7.384,148.360
C02761=1204.925,312.836,-69.906,-176.441,7.381,148.360
C02762=1204.930,312.588,-69.875,-176.443,7.378,148.360
C02763=1204.934,312.341,-69.845,-176.445,7.375,148.359
C02764=1204.938,312.091,-69.814,-176.448,7.373,148.360
C02765=1204.942,311.844,-69.784,-176.450,7.370,148.360
C02766=1204.946,311.596,-69.754,-176.452,7.368,148.360
C02767=1204.950,311.348,-69.723,-176.455,7.365,148.360
C02768=1204.955,311.099,-69.693,-176.457,7.361,148.359
C02769=1204.960,310.852,-69.663,-176.459,7.359,148.359
C02770=1204.963,310.603,-69.632,-176.462,7.356,148.359
C02771=1204.968,310.355,-69.602,-176.464,7.354,148.360
C02772=1204.972,310.107,-69.572,-176.467,7.351,148.360
C02773=1204.977,309.859,-69.541,-176.470,7.348,148.360
C02774=1204.981,309.611,-69.512,-176.472,7.346,148.360
C02775=1204.985,309.363,-69.481,-176.474,7.342,148.359
C02776=1204.989,309.114,-69.451,-176.477,7.339,148.359
C02777=1204.993,308.866,-69.420,-176.479,7.337,148.359
C02778=1204.997,308.618,-69.390,-176.481,7.334,148.359
C02779=1205.002,308.370,-69.361,-176.484,7.332,148.360
C02780=1205.006,308.122,-69.330,-176.486,7.329,148.360
C02781=1205.010,307.874,-69.300,-176.489,7.326,148.360
C02782=1205.015,307.626,-69.270,-176.491,7.323,148.360
C02783=1205.019,307.377,-69.240,-176.494,7.320,148.360
C02784=1205.024,307.130,-69.209,-176.495,7.318,148.359
C02785=1205.028,306.881,-69.180,-176.498,7.315,148.359
C02786=1205.031,306.633,-69.149,-176.501,7.312,148.359
C02787=1205.036,306.384,-69.119,-176.503,7.310,148.360
C02788=1205.040,306.137,-69.089,-176.506,7.307,148.360
C02789=1205.045,305.888,-69.059,-176.508,7.304,148.360
C02790=1205.049,305.640,-69.029,-176.510,7.301,148.360
C02791=1205.053,305.392,-69.000,-176.513,7.298,148.360
C02792=1205.058,305.144,-68.969,-176.515,7.296,148.360
C02793=1205.062,304.896,-68.939,-176.518,7.293,148.360
C02794=1205.066,304.648,-68.910,-176.520,7.291,148.360
C02795=1205.071,304.400,-68.879,-176.523,7.288,148.360
C02796=1205.075,304.151,-68.850,-176.525,7.285,148.360
C02797=1205.079,303.903,-68.820,-176.528,7.283,148.360
C02798=1205.084,303.655,-68.789,-176.530,7.280,148.360
C02799=1205.088,303.407,-68.760,-176.532,7.277,148.360
C02800=1205.092,303.159,-68.731,-176.535,7.274,148.360
C02801=1205.096,302.911,-68.700,-176.537,7.271,148.360
C02802=1205.101,302.662,-68.670,-176.539,7.269,148.360
C02803=1205.105,302.414,-68.641,-176.542,7.266,148.360
C02804=1205.109,302.166,-68.611,-176.544,7.264,148.360
C02805=1205.113,301.918,-68.581,-176.547,7.261,148.360
C02806=1205.118,301.670,-68.551,-176.549,7.259,148.360
C02807=1205.122,301.421,-68.522,-176.552,7.256,148.360
C02808=1205.126,301.173,-68.492,-176.554,7.252,148.360
C02809=1205.130,300.926,-68.462,-176.557,7.250,148.360
C02810=1205.135,300.677,-68.432,-176.559,7.247,148.360
C02811=1205.139,300.429,-68.403,-176.561,7.245,148.360
C02812=1205.143,300.180,-68.373,-176.564,7.242,148.360
C02813=1205.148,299.932,-68.344,-176.566,7.240,148.360
C02814=1205.152,299.684,-68.314,-176.569,7.237,148.360
C02815=1205.156,299.436,-68.285,-176.572,7.234,148.360
C02816=1205.161,299.188,-68.254,-176.574,7.232,148.360
C02817=1205.165,298.939,-68.225,-176.576,7.229,148.360
C02818=1205.169,298.691,-68.195,-176.579,7.226,148.360
C02819=1205.173,298.443,-68.166,-176.582,7.224,148.361
C02820=1205.177,298.195,-68.136,-176.584,7.221,148.361
C02821=1205.182,297.947,-68.107,-176.586,7.218,148.361
C02822=1205.186,297.699,-68.078,-176.589,7.215,148.361
C02823=1205.190,297.450,-68.048,-176.591,7.213,148.361
C02824=1205.195,297.202,-68.018,-176.594,7.210,148.361
C02825=1205.200,296.954,-67.989,-176.596,7.208,148.361
C02826=1205.204,296.705,-67.959,-176.599,7.205,148.361
C02827=1205.208,296.457,-67.930,-176.601,7.203,148.361
C02828=1205.212,296.209,-67.900,-176.604,7.200,148.361
C02829=1205.216,295.961,-67.871,-176.606,7.198,148.361
C02830=1205.220,295.712,-67.841,-176.608,7.195,148.361
C02831=1205.225,295.465,-67.812,-176.611,7.192,148.361
C02832=1205.229,295.216,-67.783,-176.613,7.189,148.361
C02833=1205.234,294.968,-67.753,-176.616,7.186,148.361
C02834=1205.238,294.720,-67.724,-176.618,7.184,148.361
C02835=1205.242,294.472,-67.695,-176.621,7.181,148.361
C02836=1205.246,294.223,-67.666,-176.623,7.179,148.361
C02837=1205.251,293.975,-67.636,-176.626,7.176,148.361
C02838=1205.255,293.727,-67.607,-176.628,7.174,148.362
C02839=1205.260,293.479,-67.578,-176.631,7.171,148.362
C02840=1205.264,293.230,-67.548,-176.634,7.168,148.362
C02841=1205.268,292.982,-67.519,-176.636,7.166,148.362
C02842=1205.272,292.733,-67.490,-176.638,7.163,148.362
C02843=1205.277,292.485,-67.461,-176.641,7.161,148.362
C02844=1205.281,292.237,-67.432,-176.644,7.158,148.362
C02845=1205.286,291.989,-67.402,-176.646,7.156,148.362
C02846=1205.289,291.741,-67.374,-176.649,7.153,148.362
C02847=1205.293,291.492,-67.345,-176.651,7.150,148.362
C02848=1205.298,291.244,-67.315,-176.653,7.147,148.362
C02849=1205.302,290.996,-67.286,-176.656,7.145,148.362
C02850=1205.307,290.748,-67.257,-176.658,7.142,148.362
C02851=1205.311,290.499,-67.228,-176.660,7.140,148.362
C02852=1205.315,290.251,-67.198,-176.663,7.137,148.363
C02853=1205.320,290.002,-67.170,-176.666,7.135,148.363
C02854=1205.325,289.755,-67.141,-176.668,7.132,148.363
C02855=1205.328,289.507,-67.112,-176.670,7.130,148.363
C02856=1205.334,289.232,-67.079,-176.673,7.127,148.363
C02857=1205.338,288.958,-67.048,-176.676,7.124,148.363
C02858=1205.343,288.684,-67.015,-176.679,7.121,148.363
C02859=1205.347,288.409,-66.983,-176.682,7.118,148.363
C02860=1205.352,288.161,-66.955,-176.684,7.115,148.363
C02861=1205.356,287.912,-66.926,-176.687,7.113,148.363
C02862=1205.361,287.664,-66.896,-176.690,7.110,148.363
C02863=1205.365,287.416,-66.868,-176.692,7.108,148.363
C02864=1205.369,287.168,-66.839,-176.695,7.105,148.363
C02865=1205.374,286.919,-66.810,-176.697,7.103,148.364
C02866=1205.378,286.671,-66.781,-176.700,7.100,148.364
C02867=1205.382,286.423,-66.753,-176.702,7.098,148.364
C02868=1205.386,286.175,-66.724,-176.705,7.095,148.364
C02869=1205.391,285.926,-66.695,-176.707,7.093,148.364
C02870=1205.396,285.678,-66.666,-176.709,7.090,148.364
C02871=1205.399,285.430,-66.638,-176.712,7.088,148.364
C02872=1205.404,285.181,-66.609,-176.715,7.085,148.364
C02873=1205.409,284.933,-66.580,-176.717,7.083,148.364
C02874=1205.412,284.685,-66.552,-176.720,7.080,148.364
C02875=1205.416,284.436,-66.522,-176.722,7.077,148.364
C02876=1205.422,284.188,-66.494,-176.725,7.075,148.365
C02877=1205.425,283.940,-66.466,-176.727,7.073,148.365
C02878=1205.429,283.691,-66.436,-176.729,7.070,148.365
C02879=1205.435,283.443,-66.408,-176.732,7.067,148.365
C02880=1205.438,283.195,-66.380,-176.734,7.065,148.365
C02881=1205.443,282.946,-66.350,-176.737,7.062,148.365
C02882=1205.448,282.698,-66.322,-176.739,7.060,148.365
C02883=1205.451,282.449,-66.294,-176.742,7.057,148.365
C02884=1205.456,282.202,-66.265,-176.744,7.055,148.365
C02885=1205.461,281.953,-66.236,-176.747,7.052,148.366
C02886=1205.464,281.704,-66.208,-176.749,7.050,148.366
C02887=1205.469,281.456,-66.179,-176.752,7.047,148.366
C02888=1205.473,281.208,-66.151,-176.754,7.045,148.366
C02889=1205.478,280.960,-66.122,-176.757,7.042,148.366
C02890=1205.482,280.712,-66.094,-176.760,7.040,148.366
C02891=1205.486,280.463,-66.065,-176.762,7.037,148.366
C02892=1205.491,280.214,-66.037,-176.764,7.035,148.366
C02893=1205.495,279.967,-66.008,-176.768,7.032,148.366
C02894=1205.500,279.718,-65.980,-176.770,7.030,148.367
C02895=1205.504,279.470,-65.952,-176.772,7.027,148.367
C02896=1205.509,279.222,-65.923,-176.775,7.025,148.367
C02897=1205.512,278.973,-65.895,-176.777,7.023,148.367
C02898=1205.517,278.724,-65.866,-176.780,7.020,148.367
C02899=1205.521,278.476,-65.838,-176.782,7.018,148.367
C02900=1205.526,278.227,-65.810,-176.785,7.015,148.367
C02901=1205.530,277.980,-65.781,-176.787,7.013,148.367
C02902=1205.534,277.731,-65.753,-176.790,7.010,148.367
C02903=1205.539,277.483,-65.725,-176.793,7.008,148.368
C02904=1205.543,277.234,-65.696,-176.795,7.005,148.368
C02905=1205.547,276.987,-65.668,-176.797,7.003,148.368
C02906=1205.551,276.738,-65.640,-176.800,7.000,148.368
C02907=1205.556,276.490,-65.612,-176.803,6.998,148.368
C02908=1205.560,276.241,-65.584,-176.805,6.996,148.368
C02909=1205.565,275.993,-65.555,-176.808,6.993,148.368
C02910=1205.569,275.744,-65.527,-176.810,6.991,148.368
C02911=1205.573,275.497,-65.499,-176.813,6.988,148.369
C02912=1205.578,275.248,-65.471,-176.815,6.986,148.369
C02913=1205.582,275.000,-65.443,-176.818,6.983,148.369
C02914=1205.587,274.750,-65.415,-176.820,6.981,148.369
C02915=1205.591,274.502,-65.387,-176.822,6.978,148.369
C02916=1205.595,274.254,-65.359,-176.826,6.976,148.369
C02917=1205.600,274.006,-65.330,-176.828,6.974,148.369
C02918=1205.604,273.757,-65.302,-176.830,6.971,148.369
C02919=1205.608,273.509,-65.275,-176.833,6.969,148.370
C02920=1205.613,273.260,-65.246,-176.835,6.966,148.370
C02921=1205.617,273.012,-65.218,-176.838,6.963,148.370
C02922=1205.622,272.764,-65.191,-176.841,6.962,148.370
C02923=1205.626,272.515,-65.162,-176.843,6.959,148.370
C02924=1205.631,272.267,-65.134,-176.845,6.956,148.370
C02925=1205.634,272.019,-65.106,-176.849,6.954,148.370
C02926=1205.639,271.770,-65.078,-176.851,6.952,148.371
C02927=1205.643,271.521,-65.050,-176.853,6.949,148.371
C02928=1205.648,271.273,-65.023,-176.856,6.947,148.371
C02929=1205.652,271.026,-64.995,-176.858,6.944,148.371
C02930=1205.657,270.777,-64.966,-176.861,6.942,148.371
C02931=1205.661,270.528,-64.939,-176.863,6.940,148.371
C02932=1205.665,270.280,-64.911,-176.866,6.937,148.371
C02933=1205.669,270.032,-64.883,-176.869,6.935,148.372
C02934=1205.675,269.783,-64.856,-176.871,6.932,148.372
C02935=1205.678,269.534,-64.827,-176.874,6.929,148.372
C02936=1205.683,269.286,-64.800,-176.876,6.928,148.372
C02937=1205.688,269.038,-64.773,-176.878,6.925,148.372
C02938=1205.691,268.789,-64.744,-176.882,6.923,148.372
C02939=1205.696,268.541,-64.716,-176.884,6.921,148.372
C02940=1205.700,268.292,-64.689,-176.886,6.918,148.372
C02941=1205.705,268.044,-64.661,-176.889,6.916,148.373
C02942=1205.709,267.796,-64.634,-176.891,6.913,148.373
C02943=1205.713,267.547,-64.606,-176.894,6.910,148.373
C02944=1205.718,267.299,-64.579,-176.896,6.909,148.373
C02945=1205.723,267.050,-64.550,-176.899,6.906,148.373
C02946=1205.727,266.802,-64.522,-176.902,6.904,148.374
C02947=1205.731,266.553,-64.495,-176.904,6.902,148.374
C02948=1205.736,266.305,-64.467,-176.907,6.899,148.374
C02949=1205.740,266.057,-64.440,-176.909,6.897,148.374
C02950=1205.744,265.808,-64.412,-176.911,6.894,148.374
C02951=1205.749,265.560,-64.385,-176.915,6.892,148.374
C02952=1205.753,265.312,-64.357,-176.917,6.890,148.374
C02953=1205.757,265.063,-64.330,-176.919,6.888,148.375
C02954=1205.763,264.814,-64.302,-176.922,6.885,148.375
C02955=1205.767,264.566,-64.274,-176.924,6.883,148.375
C02956=1205.772,264.318,-64.247,-176.927,6.881,148.375
C02957=1205.775,264.069,-64.219,-176.929,6.878,148.375
C02958=1205.780,263.820,-64.192,-176.932,6.876,148.375
C02959=1205.785,263.572,-64.165,-176.935,6.873,148.375
C02960=1205.789,263.299,-64.135,-176.937,6.871,148.376
C02961=1205.794,263.026,-64.105,-176.940,6.868,148.376
C02962=1205.799,262.754,-64.074,-176.943,6.865,148.376
C02963=1205.804,262.481,-64.045,-176.945,6.863,148.376
C02964=1205.808,262.232,-64.017,-176.949,6.860,148.376
C02965=1205.812,261.984,-63.989,-176.951,6.858,148.377
C02966=1205.817,261.736,-63.962,-176.953,6.856,148.377
C02967=1205.821,261.487,-63.935,-176.956,6.853,148.377
C02968=1205.826,261.239,-63.907,-176.959,6.851,148.377
C02969=1205.830,260.990,-63.880,-176.961,6.849,148.377
C02970=1205.834,260.742,-63.853,-176.964,6.847,148.378
C02971=1205.839,260.493,-63.826,-176.966,6.844,148.378
C02972=1205.843,260.245,-63.798,-176.969,6.843,148.378
C02973=1205.847,259.996,-63.771,-176.971,6.840,148.378
C02974=1205.851,259.748,-63.744,-176.974,6.838,148.378
C02975=1205.856,259.500,-63.717,-176.976,6.835,148.378
C02976=1205.861,259.251,-63.690,-176.979,6.832,148.378
C02977=1205.865,259.003,-63.663,-176.982,6.831,148.379
C02978=1205.870,258.755,-63.635,-176.984,6.828,148.379
C02979=1205.874,258.505,-63.608,-176.987,6.826,148.379
C02980=1205.878,258.257,-63.581,-176.989,6.824,148.379
C02981=1205.883,258.008,-63.554,-176.992,6.822,148.379
C02982=1205.887,257.760,-63.527,-176.994,6.820,148.380
C02983=1205.892,257.512,-63.500,-176.997,6.817,148.380
C02984=1205.896,257.263,-63.473,-176.999,6.815,148.380
C02985=1205.901,257.015,-63.446,-177.002,6.813,148.380
C02986=1205.905,256.766,-63.419,-177.004,6.810,148.380
C02987=1205.909,256.518,-63.391,-177.007,6.808,148.381
C02988=1205.913,256.270,-63.364,-177.009,6.806,148.381
C02989=1205.918,256.021,-63.337,-177.012,6.803,148.381
C02990=1205.923,255.773,-63.310,-177.014,6.801,148.381
C02991=1205.927,255.524,-63.283,-177.017,6.799,148.381
C02992=1205.932,255.276,-63.256,-177.019,6.797,148.381
C02993=1205.936,255.027,-63.230,-177.022,6.794,148.382
C02994=1205.940,254.778,-63.202,-177.025,6.792,148.382
C02995=1205.945,254.529,-63.176,-177.027,6.790,148.382
C02996=1205.949,254.281,-63.149,-177.030,6.787,148.382
C02997=1205.953,254.032,-63.122,-177.033,6.785,148.382
C02998=1205.958,253.784,-63.095,-177.035,6.783,148.382
C02999=1205.963,253.535,-63.068,-177.038,6.780,148.383
C03000=1205.967,253.287,-63.042,-177.040,6.779,148.383
C03001=1205.971,253.039,-63.015,-177.043,6.776,148.383
C03002=1205.976,252.790,-62.988,-177.045,6.774,148.383
C03003=1205.980,252.542,-62.961,-177.048,6.771,148.384
C03004=1205.985,252.294,-62.934,-177.051,6.770,148.384
C03005=1205.989,252.044,-62.908,-177.053,6.767,148.384
C03006=1205.994,251.796,-62.881,-177.055,6.766,148.384
C03007=1205.998,251.548,-62.854,-177.058,6.763,148.384
C03008=1206.003,251.299,-62.827,-177.061,6.761,148.385
C03009=1206.007,251.051,-62.801,-177.063,6.759,148.385
C03010=1206.012,250.802,-62.774,-177.066,6.756,148.385
C03011=1206.016,250.553,-62.747,-177.069,6.754,148.385
C03012=1206.020,250.305,-62.721,-177.071,6.752,148.385
C03013=1206.025,250.057,-62.694,-177.073,6.750,148.386
C03014=1206.030,249.808,-62.668,-177.076,6.747,148.386
C03015=1206.034,249.559,-62.641,-177.079,6.745,148.386
C03016=1206.038,249.311,-62.614,-177.081,6.743,148.386
C03017=1206.042,249.063,-62.588,-177.083,6.741,148.386
C03018=1206.047,248.814,-62.561,-177.086,6.738,148.386
C03019=1206.051,248.566,-62.535,-177.089,6.736,148.387
C03020=1206.056,248.317,-62.508,-177.091,6.734,148.387
C03021=1206.061,248.068,-62.481,-177.094,6.732,148.387
C03022=1206.065,247.820,-62.455,-177.097,6.730,148.387
C03023=1206.069,247.571,-62.428,-177.099,6.727,148.388
C03024=1206.074,247.322,-62.402,-177.102,6.725,148.388
C03025=1206.078,247.074,-62.375,-177.104,6.723,148.388
C03026=1206.082,246.825,-62.349,-177.107,6.721,148.388
C03027=1206.087,246.577,-62.322,-177.110,6.719,148.389
C03028=1206.091,246.328,-62.296,-177.112,6.717,148.389
C03029=1206.096,246.079,-62.269,-177.114,6.715,148.389
C03030=1206.100,245.831,-62.243,-177.116,6.713,148.389
C03031=1206.105,245.582,-62.217,-177.120,6.710,148.389
C03032=1206.109,245.334,-62.190,-177.122,6.708,148.390
C03033=1206.114,245.085,-62.164,-177.124,6.706,148.390
C03034=1206.118,244.837,-62.137,-177.127,6.704,148.390
C03035=1206.122,244.588,-62.112,-177.130,6.701,148.390
C03036=1206.127,244.340,-62.085,-177.132,6.699,148.390
C03037=1206.131,244.091,-62.059,-177.135,6.697,148.391
C03038=1206.136,243.843,-62.032,-177.137,6.695,148.391
C03039=1206.140,243.594,-62.006,-177.140,6.693,148.391
C03040=1206.144,243.345,-61.980,-177.143,6.691,148.391
C03041=1206.149,243.097,-61.953,-177.145,6.688,148.392
C03042=1206.153,242.848,-61.928,-177.148,6.687,148.392
C03043=1206.158,242.599,-61.901,-177.150,6.684,148.392
C03044=1206.163,242.351,-61.875,-177.153,6.682,148.392
C03045=1206.167,242.102,-61.849,-177.156,6.680,148.393
C03046=1206.172,241.854,-61.822,-177.158,6.678,148.393
C03047=1206.176,241.605,-61.797,-177.160,6.676,148.393
C03048=1206.180,241.357,-61.770,-177.163,6.674,148.393
C03049=1206.185,241.108,-61.744,-177.166,6.671,148.393
C03050=1206.189,240.859,-61.718,-177.168,6.669,148.394
C03051=1206.194,240.611,-61.693,-177.171,6.667,148.394
C03052=1206.199,240.362,-61.666,-177.173,6.665,148.394
C03053=1206.203,240.114,-61.640,-177.176,6.663,148.394
C03054=1206.207,239.865,-61.614,-177.179,6.660,148.394
C03055=1206.212,239.616,-61.587,-177.181,6.658,148.395
C03056=1206.216,239.368,-61.562,-177.184,6.657,148.395
C03057=1206.221,239.119,-61.536,-177.186,6.654,148.395
C03058=1206.225,238.870,-61.510,-177.189,6.653,148.395
C03059=1206.230,238.622,-61.483,-177.191,6.651,148.396
C03060=1206.234,238.373,-61.457,-177.194,6.648,148.396
C03061=1206.239,238.125,-61.432,-177.197,6.646,148.396
C03062=1206.243,237.876,-61.406,-177.199,6.644,148.396
C03063=1206.248,237.627,-61.380,-177.201,6.642,148.397
C03064=1206.252,237.356,-61.351,-177.205,6.639,148.397
C03065=1206.257,237.085,-61.323,-177.207,6.637,148.397
C03066=1206.262,236.813,-61.295,-177.210,6.635,148.397
C03067=1206.267,236.542,-61.267,-177.213,6.633,148.398
C03068=1206.271,236.293,-61.241,-177.215,6.631,148.398
C03069=1206.276,236.044,-61.215,-177.218,6.629,148.398
C03070=1206.281,235.795,-61.189,-177.221,6.626,148.398
C03071=1206.285,235.547,-61.164,-177.223,6.624,148.399
C03072=1206.290,235.299,-61.138,-177.226,6.622,148.399
C03073=1206.294,235.050,-61.112,-177.228,6.620,148.399
C03074=1206.298,234.801,-61.087,-177.231,6.618,148.399
C03075=1206.303,234.553,-61.061,-177.233,6.616,148.400
C03076=1206.308,234.304,-61.035,-177.236,6.614,148.400
C03077=1206.312,234.055,-61.009,-177.239,6.611,148.400
C03078=1206.316,233.806,-60.983,-177.241,6.609,148.400
C03079=1206.321,233.558,-60.958,-177.244,6.608,148.401
C03080=1206.325,233.309,-60.932,-177.246,6.606,148.401
C03081=1206.330,233.060,-60.906,-177.249,6.604,148.401
C03082=1206.334,232.812,-60.881,-177.251,6.602,148.401
C03083=1206.339,232.564,-60.855,-177.254,6.599,148.402
C03084=1206.343,232.315,-60.830,-177.257,6.597,148.402
C03085=1206.348,232.067,-60.804,-177.259,6.595,148.402
C03086=1206.353,231.817,-60.778,-177.262,6.593,148.402
C03087=1206.357,231.569,-60.752,-177.264,6.591,148.403
C03088=1206.362,231.321,-60.727,-177.267,6.589,148.403
C03089=1206.366,231.072,-60.701,-177.269,6.587,148.403
C03090=1206.370,230.822,-60.676,-177.272,6.585,148.403
C03091=1206.375,230.574,-60.651,-177.275,6.583,148.404
C03092=1206.380,230.325,-60.625,-177.277,6.581,148.404
C03093=1206.384,230.077,-60.599,-177.280,6.579,148.404
C03094=1206.389,229.829,-60.574,-177.282,6.577,148.405
C03095=1206.393,229.580,-60.548,-177.285,6.575,148.405
C03096=1206.398,229.331,-60.523,-177.287,6.573,148.405
C03097=1206.402,229.082,-60.497,-177.290,6.570,148.405
C03098=1206.406,228.833,-60.472,-177.293,6.568,148.406
C03099=1206.410,228.586,-60.447,-177.295,6.566,148.406
C03100=1206.415,228.336,-60.422,-177.298,6.564,148.406
C03101=1206.420,228.088,-60.396,-177.301,6.563,148.406
C03102=1206.424,227.839,-60.371,-177.303,6.561,148.407
C03103=1206.428,227.590,-60.345,-177.305,6.559,148.407
C03104=1206.433,227.342,-60.320,-177.308,6.557,148.407
C03105=1206.438,227.093,-60.295,-177.311,6.554,148.407
C03106=1206.442,226.845,-60.269,-177.314,6.552,148.408
C03107=1206.447,226.595,-60.244,-177.316,6.550,148.408
C03108=1206.452,226.347,-60.219,-177.319,6.548,148.408
C03109=1206.456,226.099,-60.193,-177.321,6.546,148.408
C03110=1206.460,225.849,-60.169,-177.324,6.545,148.409
C03111=1206.465,225.601,-60.143,-177.326,6.542,148.409
C03112=1206.469,225.352,-60.118,-177.329,6.541,148.409
C03113=1206.474,225.104,-60.093,-177.331,6.539,148.410
C03114=1206.478,224.855,-60.067,-177.334,6.536,148.410
C03115=1206.483,224.606,-60.042,-177.337,6.534,148.410
C03116=1206.488,224.357,-60.017,-177.339,6.532,148.410
C03117=1206.492,224.109,-59.993,-177.342,6.530,148.411
C03118=1206.496,223.860,-59.967,-177.345,6.528,148.411
C03119=1206.501,223.611,-59.942,-177.347,6.527,148.411
C03120=1206.506,223.363,-59.916,-177.349,6.524,148.411
C03121=1206.511,223.114,-59.892,-177.352,6.523,148.412
C03122=1206.514,222.865,-59.867,-177.355,6.521,148.412
C03123=1206.519,222.617,-59.842,-177.357,6.519,148.412
C03124=1206.524,222.368,-59.816,-177.360,6.516,148.413
C03125=1206.529,222.119,-59.791,-177.363,6.514,148.413
C03126=1206.532,221.871,-59.766,-177.365,6.512,148.413
C03127=1206.537,221.622,-59.742,-177.368,6.510,148.413
C03128=1206.542,221.373,-59.716,-177.371,6.508,148.414
C03129=1206.547,221.124,-59.691,-177.373,6.507,148.414
C03130=1206.550,220.875,-59.667,-177.375,6.504,148.414
C03131=1206.555,220.627,-59.641,-177.378,6.503,148.415
C03132=1206.560,220.378,-59.616,-177.381,6.501,148.415
C03133=1206.564,220.130,-59.592,-177.383,6.499,148.415
C03134=1206.568,219.881,-59.567,-177.386,6.497,148.416
C03135=1206.574,219.632,-59.542,-177.389,6.495,148.416
C03136=1206.578,219.384,-59.517,-177.391,6.492,148.416
C03137=1206.582,219.135,-59.492,-177.394,6.490,148.416
C03138=1206.587,218.886,-59.467,-177.397,6.489,148.417
C03139=1206.591,218.637,-59.442,-177.399,6.487,148.417
C03140=1206.596,218.389,-59.418,-177.402,6.485,148.417
C03141=1206.600,218.139,-59.392,-177.404,6.483,148.417
C03142=1206.605,217.891,-59.368,-177.407,6.481,148.418
C03143=1206.610,217.643,-59.343,-177.409,6.479,148.418
C03144=1206.614,217.393,-59.318,-177.412,6.477,148.418
C03145=1206.619,217.145,-59.294,-177.415,6.475,148.419
C03146=1206.623,216.896,-59.269,-177.417,6.474,148.419
C03147=1206.627,216.648,-59.244,-177.420,6.472,148.419
C03148=1206.632,216.399,-59.219,-177.422,6.470,148.419
C03149=1206.637,216.150,-59.194,-177.425,6.467,148.420
C03150=1206.641,215.901,-59.170,-177.428,6.465,148.420
C03151=1206.646,215.652,-59.146,-177.430,6.463,148.420
C03152=1206.650,215.404,-59.120,-177.433,6.461,148.421
C03153=1206.655,215.155,-59.096,-177.436,6.460,148.421
C03154=1206.659,214.906,-59.071,-177.438,6.458,148.421
C03155=1206.664,214.657,-59.047,-177.441,6.456,148.422
C03156=1206.668,214.409,-59.023,-177.443,6.454,148.422
C03157=1206.673,214.160,-58.998,-177.446,6.452,148.422
C03158=1206.677,213.911,-58.974,-177.448,6.450,148.423
C03159=1206.682,213.662,-58.949,-177.451,6.448,148.423
C03160=1206.686,213.413,-58.924,-177.454,6.446,148.423
C03161=1206.691,213.165,-58.899,-177.456,6.445,148.424
C03162=1206.695,212.917,-58.875,-177.459,6.442,148.424
C03163=1206.700,212.667,-58.850,-177.461,6.441,148.424
C03164=1206.704,212.419,-58.826,-177.464,6.439,148.424
C03165=1206.709,212.170,-58.801,-177.466,6.437,148.425
C03166=1206.714,211.922,-58.777,-177.469,6.435,148.425
C03167=1206.718,211.672,-58.752,-177.472,6.432,148.425
C03168=1206.724,211.402,-58.726,-177.475,6.431,148.426
C03169=1206.728,211.132,-58.700,-177.478,6.429,148.426
C03170=1206.733,210.862,-58.673,-177.480,6.427,148.426
C03171=1206.738,210.591,-58.646,-177.483,6.424,148.427
C03172=1206.742,210.342,-58.622,-177.486,6.422,148.427
C03173=1206.747,210.094,-58.597,-177.489,6.421,148.427
C03174=1206.752,209.845,-58.574,-177.491,6.419,148.428
C03175=1206.757,209.595,-58.549,-177.494,6.417,148.428
C03176=1206.761,209.347,-58.525,-177.497,6.415,148.428
C03177=1206.766,209.098,-58.501,-177.499,6.413,148.428
C03178=1206.771,208.850,-58.476,-177.501,6.411,148.429
C03179=1206.774,208.600,-58.452,-177.504,6.409,148.429
C03180=1206.779,208.352,-58.428,-177.507,6.407,148.429
C03181=1206.784,208.103,-58.403,-177.509,6.406,148.430
C03182=1206.789,207.854,-58.380,-177.512,6.404,148.430
C03183=1206.793,207.606,-58.356,-177.515,6.402,148.430
C03184=1206.798,207.356,-58.331,-177.517,6.400,148.431
C03185=1206.802,207.108,-58.306,-177.520,6.398,148.431
C03186=1206.806,206.860,-58.282,-177.523,6.396,148.431
C03187=1206.812,206.610,-58.258,-177.525,6.395,148.432
C03188=1206.816,206.362,-58.234,-177.527,6.393,148.432
C03189=1206.820,206.113,-58.210,-177.530,6.391,148.432
C03190=1206.825,205.864,-58.185,-177.533,6.389,148.433
C03191=1206.830,205.615,-58.162,-177.535,6.387,148.433
C03192=1206.834,205.367,-58.138,-177.538,6.385,148.433
C03193=1206.839,205.118,-58.114,-177.541,6.383,148.434
C03194=1206.843,204.868,-58.089,-177.543,6.382,148.434
C03195=1206.848,204.620,-58.065,-177.546,6.380,148.434
C03196=1206.852,204.371,-58.041,-177.549,6.378,148.435
C03197=1206.857,204.122,-58.018,-177.551,6.376,148.435
C03198=1206.861,203.874,-57.994,-177.554,6.374,148.435
C03199=1206.866,203.625,-57.969,-177.557,6.372,148.436
C03200=1206.871,203.376,-57.946,-177.559,6.371,148.436
C03201=1206.875,203.127,-57.921,-177.562,6.369,148.436
C03202=1206.880,202.878,-57.898,-177.565,6.367,148.437
C03203=1206.884,202.630,-57.874,-177.567,6.365,148.437
C03204=1206.889,202.381,-57.849,-177.569,6.363,148.437
C03205=1206.894,202.132,-57.826,-177.572,6.361,148.437
C03206=1206.898,201.883,-57.802,-177.575,6.359,148.438
C03207=1206.903,201.634,-57.778,-177.577,6.357,148.438
C03208=1206.907,201.386,-57.754,-177.580,6.356,148.439
C03209=1206.911,201.136,-57.731,-177.583,6.354,148.439
C03210=1206.916,200.888,-57.707,-177.585,6.352,148.439
C03211=1206.921,200.639,-57.683,-177.588,6.350,148.440
C03212=1206.926,200.390,-57.659,-177.591,6.348,148.440
C03213=1206.930,200.141,-57.635,-177.593,6.346,148.440
C03214=1206.935,199.893,-57.611,-177.595,6.345,148.441
C03215=1206.939,199.644,-57.588,-177.598,6.344,148.441
C03216=1206.944,199.395,-57.564,-177.601,6.342,148.441
C03217=1206.949,199.146,-57.540,-177.603,6.340,148.442
C03218=1206.953,198.898,-57.516,-177.606,6.338,148.442
C03219=1206.958,198.649,-57.493,-177.608,6.336,148.442
C03220=1206.962,198.400,-57.470,-177.611,6.335,148.443
C03221=1206.967,198.151,-57.445,-177.614,6.333,148.443
C03222=1206.971,197.902,-57.422,-177.616,6.331,148.443
C03223=1206.976,197.654,-57.398,-177.619,6.329,148.444
C03224=1206.980,197.404,-57.374,-177.622,6.327,148.444
C03225=1206.985,197.155,-57.351,-177.624,6.325,148.444
C03226=1206.989,196.907,-57.327,-177.627,6.324,148.445
C03227=1206.994,196.658,-57.304,-177.630,6.322,148.445
C03228=1206.998,196.409,-57.280,-177.632,6.320,148.445
C03229=1207.003,196.160,-57.256,-177.635,6.318,148.446
C03230=1207.008,195.911,-57.233,-177.638,6.316,148.446
C03231=1207.012,195.662,-57.209,-177.640,6.314,148.446
C03232=1207.017,195.413,-57.186,-177.642,6.313,148.447
C03233=1207.021,195.165,-57.162,-177.645,6.312,148.447
C03234=1207.026,194.916,-57.139,-177.648,6.310,148.448
C03235=1207.031,194.667,-57.115,-177.650,6.308,148.448
C03236=1207.035,194.417,-57.092,-177.653,6.306,148.448
C03237=1207.040,194.170,-57.068,-177.656,6.304,148.449
C03238=1207.045,193.921,-57.045,-177.658,6.303,148.449
C03239=1207.050,193.672,-57.021,-177.661,6.301,148.449
C03240=1207.055,193.423,-56.998,-177.664,6.299,148.450
C03241=1207.059,193.174,-56.975,-177.666,6.297,148.450
C03242=1207.064,192.925,-56.951,-177.669,6.295,148.450
C03243=1207.068,192.677,-56.928,-177.672,6.293,148.451
C03244=1207.072,192.428,-56.905,-177.674,6.292,148.451
C03245=1207.077,192.178,-56.881,-177.676,6.291,148.451
C03246=1207.082,191.929,-56.858,-177.679,6.289,148.452
C03247=1207.086,191.680,-56.834,-177.682,6.287,148.452
C03248=1207.091,191.431,-56.811,-177.684,6.285,148.452
C03249=1207.096,191.182,-56.788,-177.687,6.283,148.453
C03250=1207.100,190.934,-56.765,-177.690,6.282,148.453
C03251=1207.104,190.685,-56.742,-177.692,6.280,148.453
C03252=1207.109,190.437,-56.718,-177.695,6.278,148.454
C03253=1207.114,190.188,-56.695,-177.698,6.276,148.454
C03254=1207.119,189.939,-56.671,-177.700,6.275,148.455
C03255=1207.124,189.690,-56.648,-177.702,6.273,148.455
C03256=1207.128,189.441,-56.625,-177.705,6.271,148.455
C03257=1207.132,189.192,-56.602,-177.708,6.270,148.456
C03258=1207.137,188.943,-56.578,-177.710,6.268,148.456
C03259=1207.142,188.694,-56.555,-177.713,6.266,148.456
C03260=1207.146,188.445,-56.532,-177.716,6.264,148.457
C03261=1207.151,188.197,-56.509,-177.718,6.262,148.457
C03262=1207.156,187.947,-56.487,-177.721,6.261,148.457
C03263=1207.161,187.698,-56.463,-177.723,6.260,148.458
C03264=1207.165,187.449,-56.440,-177.726,6.258,148.458
C03265=1207.169,187.200,-56.417,-177.728,6.256,148.458
C03266=1207.174,186.951,-56.394,-177.731,6.254,148.459
C03267=1207.179,186.703,-56.371,-177.734,6.252,148.459
C03268=1207.183,186.454,-56.348,-177.736,6.250,148.460
C03269=1207.188,186.205,-56.325,-177.739,6.249,148.460
C03270=1207.193,185.956,-56.301,-177.742,6.247,148.460
C03271=1207.197,185.708,-56.279,-177.744,6.246,148.461
C03272=1207.202,185.438,-56.253,-177.747,6.244,148.461
C03273=1207.207,185.168,-56.228,-177.750,6.242,148.462
C03274=1207.212,184.899,-56.204,-177.753,6.240,148.462
C03275=1207.217,184.629,-56.179,-177.755,6.238,148.462
C03276=1207.221,184.380,-56.156,-177.758,6.236,148.463
C03277=1207.227,184.131,-56.134,-177.761,6.235,148.463
C03278=1207.231,183.882,-56.111,-177.763,6.234,148.464
C03279=1207.235,183.633,-56.088,-177.766,6.232,148.464
C03280=1207.240,183.384,-56.064,-177.769,6.230,148.464
C03281=1207.245,183.135,-56.042,-177.771,6.228,148.465
C03282=1207.250,182.887,-56.019,-177.774,6.227,148.465
C03283=1207.254,182.638,-55.996,-177.777,6.225,148.465
C03284=1207.258,182.389,-55.973,-177.779,6.224,148.466
C03285=1207.263,182.139,-55.951,-177.781,6.222,148.466
C03286=1207.268,181.891,-55.928,-177.784,6.220,148.466
C03287=1207.273,181.642,-55.905,-177.787,6.218,148.467
C03288=1207.278,181.393,-55.882,-177.789,6.216,148.467
C03289=1207.282,181.144,-55.859,-177.792,6.215,148.467
C03290=1207.287,180.896,-55.836,-177.794,6.214,148.468
C03291=1207.291,180.646,-55.814,-177.797,6.212,148.468
C03292=1207.296,180.397,-55.791,-177.800,6.210,148.469
C03293=1207.300,180.149,-55.769,-177.802,6.209,148.469
C03294=1207.305,179.900,-55.746,-177.805,6.207,148.469
C03295=1207.309,179.651,-55.723,-177.808,6.205,148.470
C03296=1207.314,179.401,-55.701,-177.810,6.204,148.470
C03297=1207.319,179.153,-55.678,-177.813,6.202,148.471
C03298=1207.324,178.903,-55.656,-177.815,6.200,148.471
C03299=1207.328,178.655,-55.633,-177.818,6.198,148.471
C03300=1207.333,178.406,-55.610,-177.821,6.197,148.472
C03301=1207.337,178.157,-55.588,-177.824,6.195,148.472
C03302=1207.342,177.908,-55.564,-177.826,6.194,148.473
C03303=1207.347,177.659,-55.543,-177.828,6.192,148.473
C03304=1207.351,177.411,-55.520,-177.831,6.191,148.473
C03305=1207.356,177.161,-55.497,-177.834,6.189,148.474
C03306=1207.361,176.913,-55.475,-177.836,6.187,148.474
C03307=1207.366,176.663,-55.452,-177.838,6.186,148.474
C03308=1207.370,176.414,-55.430,-177.841,6.184,148.475
C03309=1207.375,176.166,-55.407,-177.844,6.183,148.475
C03310=1207.379,175.916,-55.385,-177.847,6.181,148.476
C03311=1207.383,175.668,-55.362,-177.850,6.179,148.476
C03312=1207.389,175.419,-55.340,-177.852,6.178,148.476
C03313=1207.393,175.170,-55.317,-177.854,6.176,148.477
C03314=1207.398,174.920,-55.295,-177.857,6.174,148.477
C03315=1207.403,174.672,-55.273,-177.860,6.173,148.478
C03316=1207.407,174.423,-55.250,-177.862,6.171,148.478
C03317=1207.412,174.174,-55.228,-177.865,6.170,148.479
C03318=1207.417,173.925,-55.206,-177.868,6.168,148.479
C03319=1207.421,173.676,-55.183,-177.870,6.167,148.479
C03320=1207.426,173.427,-55.161,-177.873,6.165,148.480
C03321=1207.430,173.178,-55.139,-177.875,6.164,148.480
C03322=1207.435,172.930,-55.116,-177.878,6.162,148.480
C03323=1207.440,172.680,-55.094,-177.880,6.160,148.481
C03324=1207.444,172.431,-55.072,-177.884,6.159,148.481
C03325=1207.449,172.183,-55.049,-177.886,6.157,148.482
C03326=1207.453,171.933,-55.027,-177.888,6.156,148.482
C03327=1207.459,171.684,-55.005,-177.891,6.154,148.482
C03328=1207.463,171.435,-54.983,-177.894,6.152,148.483
C03329=1207.468,171.187,-54.961,-177.896,6.151,148.483
C03330=1207.473,170.937,-54.938,-177.898,6.150,148.484
C03331=1207.477,170.689,-54.916,-177.902,6.148,148.484
C03332=1207.482,170.439,-54.894,-177.904,6.146,148.484
C03333=1207.486,170.190,-54.872,-177.907,6.144,148.485
C03334=1207.491,169.942,-54.849,-177.909,6.143,148.485
C03335=1207.496,169.692,-54.827,-177.912,6.142,148.486
C03336=1207.500,169.444,-54.805,-177.914,6.140,148.486
C03337=1207.505,169.194,-54.783,-177.917,6.138,148.487
C03338=1207.510,168.946,-54.762,-177.920,6.137,148.487
C03339=1207.515,168.696,-54.739,-177.922,6.136,148.487
C03340=1207.519,168.447,-54.717,-177.925,6.134,148.488
C03341=1207.523,168.199,-54.695,-177.928,6.132,148.488
C03342=1207.528,167.950,-54.673,-177.930,6.131,148.488
C03343=1207.533,167.701,-54.651,-177.933,6.130,148.489
C03344=1207.537,167.452,-54.629,-177.935,6.128,148.489
C03345=1207.542,167.202,-54.607,-177.938,6.126,148.490
C03346=1207.547,166.954,-54.585,-177.940,6.125,148.490
C03347=1207.552,166.704,-54.563,-177.943,6.123,148.490
C03348=1207.556,166.456,-54.541,-177.946,6.121,148.491
C03349=1207.561,166.206,-54.519,-177.949,6.120,148.491
C03350=1207.566,165.958,-54.497,-177.951,6.119,148.492
C03351=1207.570,165.709,-54.476,-177.953,6.117,148.492
C03352=1207.575,165.460,-54.454,-177.956,6.115,148.493
C03353=1207.580,165.211,-54.431,-177.959,6.113,148.493
C03354=1207.585,164.962,-54.409,-177.961,6.113,148.494
C03355=1207.589,164.713,-54.388,-177.964,6.111,148.494
C03356=1207.594,164.464,-54.366,-177.967,6.109,148.494
C03357=1207.599,164.215,-54.344,-177.969,6.108,148.495
C03358=1207.603,163.966,-54.322,-177.971,6.106,148.495
C03359=1207.608,163.717,-54.300,-177.975,6.105,148.496
C03360=1207.613,163.468,-54.279,-177.977,6.103,148.496
C03361=1207.617,163.219,-54.257,-177.979,6.102,148.496
C03362=1207.622,162.970,-54.235,-177.982,6.100,148.497
C03363=1207.626,162.720,-54.214,-177.985,6.099,148.497
C03364=1207.631,162.472,-54.192,-177.987,6.098,148.498
C03365=1207.636,162.223,-54.170,-177.990,6.096,148.498
C03366=1207.640,161.974,-54.148,-177.993,6.094,148.498
C03367=1207.645,161.725,-54.126,-177.995,6.093,148.499
C03368=1207.649,161.476,-54.104,-177.997,6.092,148.499
C03369=1207.655,161.226,-54.083,-178.001,6.090,148.500
C03370=1207.659,160.978,-54.062,-178.003,6.088,148.500
C03371=1207.664,160.728,-54.040,-178.005,6.087,148.501
C03372=1207.669,160.480,-54.018,-178.008,6.086,148.501
C03373=1207.673,160.230,-53.996,-178.011,6.084,148.501
C03374=1207.678,159.981,-53.975,-178.014,6.082,148.502
C03375=1207.683,159.733,-53.953,-178.016,6.081,148.502
C03376=1207.688,159.464,-53.931,-178.019,6.080,148.503
C03377=1207.693,159.195,-53.906,-178.022,6.078,148.503
C03378=1207.698,158.925,-53.883,-178.024,6.076,148.504
C03379=1207.703,158.656,-53.860,-178.028,6.075,148.504
C03380=1207.708,158.408,-53.839,-178.030,6.073,148.505
C03381=1207.712,158.158,-53.817,-178.032,6.072,148.505
C03382=1207.717,157.909,-53.796,-178.035,6.070,148.505
C03383=1207.722,157.661,-53.774,-178.038,6.068,148.506
C03384=1207.727,157.411,-53.752,-178.040,6.068,148.506
C03385=1207.731,157.162,-53.732,-178.043,6.066,148.507
C03386=1207.736,156.914,-53.710,-178.046,6.064,148.507
C03387=1207.740,156.664,-53.688,-178.048,6.063,148.508
C03388=1207.745,156.415,-53.667,-178.051,6.062,148.508
C03389=1207.750,156.166,-53.645,-178.054,6.060,148.508
C03390=1207.754,155.917,-53.623,-178.056,6.059,148.509
C03391=1207.760,155.668,-53.602,-178.058,6.057,148.509
C03392=1207.764,155.419,-53.581,-178.062,6.056,148.510
C03393=1207.769,155.170,-53.560,-178.064,6.055,148.510
C03394=1207.773,154.921,-53.538,-178.066,6.053,148.511
C03395=1207.778,154.672,-53.517,-178.069,6.051,148.511
C03396=1207.783,154.423,-53.495,-178.072,6.051,148.512
C03397=1207.788,154.174,-53.475,-178.074,6.049,148.512
C03398=1207.792,153.925,-53.453,-178.077,6.047,148.512
C03399=1207.797,153.675,-53.432,-178.079,6.046,148.513
C03400=1207.802,153.427,-53.410,-178.082,6.045,148.513
C03401=1207.806,153.178,-53.390,-178.085,6.043,148.514
C03402=1207.811,152.928,-53.368,-178.087,6.042,148.514
C03403=1207.816,152.679,-53.347,-178.090,6.040,148.515
C03404=1207.821,152.431,-53.325,-178.092,6.039,148.515
C03405=1207.825,152.182,-53.305,-178.095,6.038,148.515
C03406=1207.830,151.933,-53.283,-178.098,6.036,148.516
C03407=1207.835,151.683,-53.262,-178.100,6.035,148.516
C03408=1207.839,151.434,-53.240,-178.103,6.033,148.517
C03409=1207.844,151.185,-53.220,-178.106,6.032,148.517
C03410=1207.849,150.936,-53.199,-178.108,6.031,148.518
C03411=1207.853,150.687,-53.177,-178.111,6.029,148.518
C03412=1207.858,150.438,-53.156,-178.113,6.027,148.519
C03413=1207.863,150.189,-53.135,-178.116,6.026,148.519
C03414=1207.868,149.940,-53.114,-178.119,6.025,148.520
C03415=1207.872,149.691,-53.093,-178.121,6.024,148.520
C03416=1207.877,149.442,-53.072,-178.124,6.022,148.520
C03417=1207.882,149.192,-53.050,-178.126,6.020,148.521
C03418=1207.886,148.943,-53.030,-178.129,6.020,148.521
C03419=1207.891,148.695,-53.008,-178.131,6.018,148.522
C03420=1207.896,148.446,-52.987,-178.134,6.016,148.522
C03421=1207.901,148.197,-52.967,-178.137,6.015,148.523
C03422=1207.906,147.947,-52.946,-178.139,6.014,148.523
C03423=1207.910,147.698,-52.924,-178.142,6.013,148.524
C03424=1207.914,147.449,-52.904,-178.145,6.011,148.524
C03425=1207.920,147.200,-52.883,-178.147,6.009,148.524
C03426=1207.924,146.951,-52.862,-178.149,6.009,148.525
C03427=1207.929,146.702,-52.841,-178.152,6.007,148.525
C03428=1207.933,146.453,-52.820,-178.155,6.006,148.526
C03429=1207.939,146.204,-52.799,-178.157,6.004,148.526
C03430=1207.944,145.955,-52.778,-178.160,6.003,148.527
C03431=1207.948,145.706,-52.758,-178.163,6.002,148.527
C03432=1207.952,145.456,-52.736,-178.165,6.000,148.528
C03433=1207.957,145.207,-52.715,-178.168,5.998,148.528
C03434=1207.962,144.958,-52.695,-178.171,5.998,148.529
C03435=1207.966,144.709,-52.674,-178.173,5.996,148.529
C03436=1207.972,144.460,-52.653,-178.175,5.995,148.529
C03437=1207.976,144.211,-52.633,-178.179,5.993,148.530
C03438=1207.981,143.962,-52.612,-178.181,5.993,148.530
C03439=1207.985,143.713,-52.591,-178.183,5.991,148.531
C03440=1207.991,143.464,-52.570,-178.187,5.989,148.531
C03441=1207.995,143.215,-52.549,-178.189,5.988,148.532
C03442=1208.000,142.966,-52.528,-178.191,5.987,148.532
C03443=1208.004,142.716,-52.508,-178.194,5.986,148.533
C03444=1208.009,142.467,-52.487,-178.197,5.984,148.533
C03445=1208.014,142.218,-52.466,-178.199,5.982,148.534
C03446=1208.019,141.969,-52.445,-178.202,5.982,148.534
C03447=1208.023,141.720,-52.425,-178.205,5.980,148.535
C03448=1208.028,141.471,-52.405,-178.207,5.979,148.535
C03449=1208.033,141.222,-52.384,-178.210,5.978,148.536
C03450=1208.037,140.973,-52.363,-178.212,5.977,148.536
C03451=1208.042,140.724,-52.342,-178.215,5.975,148.536
C03452=1208.047,140.475,-52.322,-178.218,5.973,148.537
C03453=1208.052,140.225,-52.301,-178.220,5.972,148.537
C03454=1208.057,139.976,-52.281,-178.223,5.971,148.538
C03455=1208.061,139.727,-52.260,-178.225,5.970,148.538
C03456=1208.066,139.478,-52.239,-178.228,5.968,148.539
C03457=1208.071,139.229,-52.219,-178.230,5.967,148.539
C03458=1208.075,138.980,-52.199,-178.233,5.966,148.540
C03459=1208.080,138.731,-52.178,-178.236,5.964,148.540
C03460=1208.085,138.481,-52.158,-178.238,5.963,148.541
C03461=1208.090,138.232,-52.137,-178.241,5.962,148.541
C03462=1208.095,137.983,-52.117,-178.243,5.961,148.542
C03463=1208.099,137.734,-52.096,-178.246,5.959,148.542
C03464=1208.104,137.485,-52.075,-178.249,5.958,148.543
C03465=1208.109,137.236,-52.055,-178.251,5.956,148.543
C03466=1208.113,136.987,-52.035,-178.253,5.955,148.543
C03467=1208.118,136.738,-52.015,-178.256,5.954,148.544
C03468=1208.123,136.488,-51.994,-178.259,5.952,148.544
C03469=1208.127,136.239,-51.974,-178.262,5.952,148.545
C03470=1208.132,135.991,-51.954,-178.264,5.950,148.545
C03471=1208.138,135.742,-51.933,-178.267,5.949,148.546
C03472=1208.142,135.492,-51.913,-178.270,5.947,148.546
C03473=1208.147,135.243,-51.893,-178.272,5.946,148.547
C03474=1208.151,134.994,-51.872,-178.275,5.945,148.547
C03475=1208.156,134.745,-51.851,-178.277,5.944,148.548
C03476=1208.161,134.496,-51.832,-178.280,5.942,148.548
C03477=1208.166,134.247,-51.811,-178.282,5.942,148.549
C03478=1208.170,133.998,-51.791,-178.285,5.940,148.549
C03479=1208.175,133.748,-51.770,-178.287,5.939,148.550
C03480=1208.180,133.480,-51.749,-178.290,5.937,148.550
C03481=1208.185,133.211,-51.726,-178.293,5.936,148.551
C03482=1208.190,132.943,-51.705,-178.296,5.934,148.551
C03483=1208.196,132.674,-51.684,-178.299,5.934,148.552
C03484=1208.200,132.425,-51.663,-178.302,5.932,148.552
C03485=1208.205,132.176,-51.643,-178.304,5.931,148.553
C03486=1208.210,131.926,-51.623,-178.307,5.929,148.553
C03487=1208.215,131.677,-51.602,-178.309,5.929,148.554
C03488=1208.219,131.428,-51.582,-178.312,5.927,148.554
C03489=1208.225,131.179,-51.563,-178.314,5.926,148.555
C03490=1208.229,130.930,-51.542,-178.317,5.924,148.555
C03491=1208.234,130.681,-51.523,-178.319,5.924,148.556
C03492=1208.239,130.431,-51.502,-178.322,5.922,148.556
C03493=1208.243,130.183,-51.481,-178.325,5.921,148.557
C03494=1208.248,129.933,-51.462,-178.327,5.920,148.557
C03495=1208.253,129.685,-51.442,-178.330,5.919,148.558
C03496=1208.258,129.435,-51.422,-178.333,5.917,148.558
C03497=1208.262,129.186,-51.401,-178.335,5.916,148.559
C03498=1208.267,128.937,-51.382,-178.338,5.915,148.559
C03499=1208.272,128.688,-51.361,-178.340,5.914,148.560
C03500=1208.276,128.438,-51.342,-178.343,5.912,148.560
C03501=1208.282,128.190,-51.321,-178.345,5.911,148.561
C03502=1208.287,127.940,-51.302,-178.348,5.910,148.561
C03503=1208.291,127.691,-51.281,-178.351,5.909,148.562
C03504=1208.296,127.441,-51.262,-178.353,5.907,148.562
C03505=1208.300,127.193,-51.241,-178.356,5.906,148.562
C03506=1208.306,126.944,-51.222,-178.359,5.905,148.563
C03507=1208.310,126.694,-51.202,-178.361,5.904,148.563
C03508=1208.315,126.445,-51.182,-178.364,5.902,148.564
C03509=1208.320,126.196,-51.162,-178.366,5.902,148.564
C03510=1208.325,125.947,-51.142,-178.369,5.900,148.565
C03511=1208.329,125.698,-51.123,-178.371,5.899,148.566
C03512=1208.334,125.448,-51.103,-178.374,5.897,148.566
C03513=1208.339,125.199,-51.082,-178.377,5.897,148.567
C03514=1208.343,124.950,-51.063,-178.379,5.895,148.567
C03515=1208.348,124.701,-51.043,-178.382,5.894,148.568
C03516=1208.353,124.452,-51.023,-178.385,5.893,148.568
C03517=1208.358,124.202,-51.004,-178.387,5.892,148.569
C03518=1208.363,123.954,-50.984,-178.390,5.890,148.569
C03519=1208.368,123.704,-50.964,-178.393,5.890,148.570
C03520=1208.372,123.455,-50.944,-178.395,5.889,148.570
C03521=1208.377,123.206,-50.924,-178.397,5.887,148.570
C03522=1208.382,122.957,-50.905,-178.400,5.886,148.571
C03523=1208.387,122.707,-50.885,-178.403,5.885,148.571
C03524=1208.391,122.458,-50.866,-178.405,5.884,148.572
C03525=1208.395,122.209,-50.845,-178.408,5.882,148.572
C03526=1208.401,121.960,-50.826,-178.411,5.882,148.573
C03527=1208.405,121.711,-50.806,-178.413,5.880,148.574
C03528=1208.410,121.461,-50.787,-178.416,5.879,148.574
C03529=1208.415,121.213,-50.767,-178.419,5.877,148.575
C03530=1208.420,120.963,-50.747,-178.421,5.876,148.575
C03531=1208.425,120.714,-50.728,-178.423,5.876,148.576
C03532=1208.430,120.465,-50.708,-178.426,5.874,148.576
C03533=1208.435,120.215,-50.689,-178.429,5.873,148.577
C03534=1208.439,119.966,-50.670,-178.431,5.872,148.577
C03535=1208.444,119.718,-50.650,-178.434,5.871,148.578
C03536=1208.449,119.468,-50.630,-178.437,5.869,148.578
C03537=1208.453,119.219,-50.610,-178.439,5.869,148.579
C03538=1208.459,118.970,-50.591,-178.442,5.867,148.579
C03539=1208.463,118.720,-50.571,-178.445,5.866,148.580
C03540=1208.467,118.471,-50.552,-178.447,5.865,148.580
C03541=1208.473,118.222,-50.533,-178.450,5.864,148.581
C03542=1208.478,117.973,-50.513,-178.452,5.863,148.581
C03543=1208.483,117.724,-50.493,-178.455,5.861,148.582
C03544=1208.487,117.475,-50.474,-178.457,5.861,148.582
C03545=1208.491,117.226,-50.455,-178.460,5.859,148.583
C03546=1208.497,116.977,-50.435,-178.463,5.858,148.583
C03547=1208.501,116.727,-50.416,-178.465,5.857,148.584
C03548=1208.506,116.478,-50.396,-178.468,5.856,148.584
C03549=1208.511,116.229,-50.377,-178.470,5.855,148.585
C03550=1208.515,115.979,-50.358,-178.473,5.853,148.585
C03551=1208.521,115.731,-50.338,-178.475,5.853,148.586
C03552=1208.526,115.481,-50.319,-178.478,5.851,148.586
C03553=1208.530,115.231,-50.299,-178.481,5.850,148.587
C03554=1208.535,114.983,-50.280,-178.483,5.850,148.587
C03555=1208.540,114.733,-50.261,-178.486,5.848,148.588
C03556=1208.545,114.485,-50.241,-178.488,5.847,148.588
C03557=1208.549,114.235,-50.222,-178.491,5.845,148.589
C03558=1208.554,113.986,-50.203,-178.494,5.845,148.589
C03559=1208.559,113.737,-50.183,-178.496,5.844,148.590
C03560=1208.564,113.487,-50.164,-178.499,5.842,148.591
C03561=1208.569,113.238,-50.146,-178.501,5.842,148.591
C03562=1208.574,112.988,-50.126,-178.504,5.840,148.592
C03563=1208.579,112.740,-50.107,-178.507,5.839,148.592
C03564=1208.583,112.490,-50.088,-178.509,5.839,148.593
C03565=1208.588,112.242,-50.068,-178.512,5.837,148.593
C03566=1208.593,111.992,-50.049,-178.514,5.836,148.594
C03567=1208.598,111.743,-50.030,-178.517,5.834,148.594
C03568=1208.603,111.493,-50.011,-178.520,5.834,148.595
C03569=1208.607,111.245,-49.992,-178.522,5.833,148.595
C03570=1208.612,110.995,-49.973,-178.525,5.831,148.596
C03571=1208.617,110.746,-49.953,-178.527,5.831,148.596
C03572=1208.621,110.497,-49.934,-178.530,5.829,148.597
C03573=1208.627,110.248,-49.915,-178.532,5.828,148.597
C03574=1208.631,109.998,-49.897,-178.535,5.828,148.598
C03575=1208.636,109.749,-49.877,-178.538,5.826,148.598
C03576=1208.641,109.500,-49.858,-178.540,5.825,148.599
C03577=1208.646,109.251,-49.839,-178.543,5.824,148.599
C03578=1208.651,109.001,-49.820,-178.546,5.823,148.600
C03579=1208.655,108.752,-49.801,-178.548,5.822,148.600
C03580=1208.660,108.503,-49.782,-178.551,5.820,148.601
C03581=1208.665,108.254,-49.763,-178.553,5.820,148.601
C03582=1208.670,108.004,-49.744,-178.556,5.819,148.602
C03583=1208.675,107.755,-49.725,-178.558,5.817,148.602
C03584=1208.679,107.487,-49.704,-178.561,5.817,148.603
C03585=1208.685,107.218,-49.684,-178.564,5.815,148.604
C03586=1208.691,106.950,-49.664,-178.567,5.815,148.604
C03587=1208.695,106.681,-49.644,-178.570,5.813,148.605
C03588=1208.700,106.433,-49.625,-178.572,5.812,148.605
C03589=1208.704,106.183,-49.606,-178.575,5.810,148.606
C03590=1208.710,105.934,-49.587,-178.577,5.810,148.606
C03591=1208.714,105.685,-49.568,-178.580,5.809,148.607
C03592=1208.720,105.435,-49.549,-178.583,5.807,148.607
C03593=1208.724,105.187,-49.531,-178.585,5.807,148.608
C03594=1208.729,104.937,-49.511,-178.588,5.806,148.609
C03595=1208.734,104.688,-49.493,-178.591,5.805,148.609
C03596=1208.739,104.438,-49.473,-178.593,5.804,148.610
C03597=1208.744,104.189,-49.455,-178.595,5.803,148.610
C03598=1208.748,103.940,-49.436,-178.598,5.801,148.611
C03599=1208.753,103.690,-49.418,-178.601,5.801,148.611
C03600=1208.759,103.441,-49.398,-178.603,5.800,148.612
C03601=1208.763,103.192,-49.379,-178.606,5.798,148.612
C03602=1208.768,102.943,-49.361,-178.608,5.797,148.613
C03603=1208.773,102.694,-49.342,-178.611,5.797,148.613
C03604=1208.777,102.444,-49.324,-178.614,5.795,148.614
C03605=1208.783,102.195,-49.304,-178.616,5.794,148.614
C03606=1208.787,101.946,-49.286,-178.619,5.794,148.615
C03607=1208.791,101.697,-49.267,-178.621,5.792,148.615
C03608=1208.797,101.448,-49.249,-178.624,5.791,148.616
C03609=1208.801,101.198,-49.230,-178.626,5.791,148.617
C03610=1208.806,100.949,-49.212,-178.629,5.789,148.617
C03611=1208.812,100.700,-49.193,-178.632,5.788,148.618
C03612=1208.816,100.450,-49.174,-178.634,5.788,148.618
C03613=1208.821,100.201,-49.156,-178.637,5.786,148.619
C03614=1208.826,99.952,-49.137,-178.639,5.785,148.619
C03615=1208.830,99.702,-49.119,-178.642,5.785,148.620
C03616=1208.835,99.453,-49.101,-178.645,5.783,148.620
C03617=1208.840,99.204,-49.081,-178.647,5.782,148.621
C03618=1208.845,98.954,-49.063,-178.650,5.781,148.621
C03619=1208.850,98.705,-49.045,-178.653,5.780,148.622
C03620=1208.855,98.456,-49.026,-178.655,5.779,148.623
C03621=1208.859,98.207,-49.007,-178.657,5.778,148.623
C03622=1208.864,97.957,-48.989,-178.661,5.777,148.624
C03623=1208.870,97.709,-48.970,-178.663,5.776,148.624
C03624=1208.875,97.459,-48.952,-178.665,5.776,148.625
C03625=1208.879,97.209,-48.934,-178.668,5.774,148.625
C03626=1208.883,96.961,-48.915,-178.671,5.773,148.626
C03627=1208.889,96.711,-48.896,-178.673,5.773,148.627
C03628=1208.893,96.462,-48.878,-178.675,5.772,148.627
C03629=1208.898,96.213,-48.859,-178.679,5.770,148.628
C03630=1208.903,95.964,-48.841,-178.681,5.769,148.628
C03631=1208.909,95.714,-48.823,-178.683,5.769,148.629
C03632=1208.913,95.464,-48.805,-178.686,5.767,148.629
C03633=1208.917,95.216,-48.786,-178.689,5.766,148.630
C03634=1208.922,94.967,-48.768,-178.691,5.766,148.630
C03635=1208.927,94.718,-48.750,-178.694,5.764,148.631
C03636=1208.932,94.467,-48.731,-178.697,5.763,148.631
C03637=1208.937,94.218,-48.713,-178.699,5.763,148.632
C03638=1208.942,93.970,-48.694,-178.701,5.762,148.633
C03639=1208.947,93.720,-48.676,-178.705,5.761,148.633
C03640=1208.951,93.471,-48.658,-178.707,5.760,148.634
C03641=1208.957,93.221,-48.639,-178.709,5.759,148.634
